  MoveL 3289 to (42.94, 64.74, -221.41) mm, rotated rx 105.8 ry 33.04 rz -145.95 deg; joints [-8.632, -27.169, 98.04, 142.565, 83.685, 20.863, -295]
  MoveL 3290 to (44.16, 62.72, -223.16) mm, rotated rx 105.8 ry 33.04 rz -145.95 deg; joints [-8.699, -27.017, 97.932, 142.503, 83.733, 20.854, -295]
  MoveL 3291 to (44.54, 61.54, -223.78) mm, rotated rx 105.8 ry 33.04 rz -145.95 deg; joints [-8.723, -26.947, 97.904, 142.483, 83.771, 20.834, -295]
  MoveL 3292 to (44.76, 60.25, -224.22) mm, rotated rx 105.8 ry 33.04 rz -145.95 deg; joints [-8.741, -26.881, 97.895, 142.469, 83.82, 20.804, -295]
  MoveL 3293 to (44.72, 57.32, -224.57) mm, rotated rx 105.8 ry 33.04 rz -145.95 deg; joints [-8.758, -26.761, 97.928, 142.462, 83.945, 20.714, -295]
  MoveL 3294 to (44.43, 54.71, -224.56) mm, rotated rx 105.8 ry 33.04 rz -145.95 deg; joints [-8.763, -26.667, 97.984, 142.467, 84.065, 20.624, -295]
  MoveL 3295 to (44.36, 54.19, -224.55) mm, rotated rx 105.8 ry 33.04 rz -145.95 deg; joints [-8.763, -26.649, 97.996, 142.469, 84.089, 20.605, -295]
  MoveL 3296 to (44.28, 53.65, -224.52) mm, rotated rx 105.8 ry 33.04 rz -145.95 deg; joints [-8.763, -26.631, 98.01, 142.471, 84.114, 20.586, -295]
  MoveL 3297 to (44.22, 53.16, -224.51) mm, rotated rx 105.8 ry 33.04 rz -145.95 deg; joints [-8.764, -26.613, 98.021, 142.472, 84.137, 20.568, -295]
  MoveL 3298 to (44.18, 52.72, -224.53) mm, rotated rx 105.8 ry 33.04 rz -145.95 deg; joints [-8.765, -26.597, 98.03, 142.472, 84.157, 20.553, -295]
  MoveL 3299 to (44.14, 52.23, -224.56) mm, rotated rx 105.8 ry 33.04 rz -145.95 deg; joints [-8.767, -26.578, 98.038, 142.472, 84.179, 20.537, -295]
  MoveL 3300 to (44.12, 51.65, -224.63) mm, rotated rx 105.8 ry 33.04 rz -145.95 deg; joints [-8.77, -26.555, 98.046, 142.471, 84.204, 20.519, -295]
  MoveL 3301 to (44.11, 51.07, -224.71) mm, rotated rx 105.8 ry 33.04 rz -145.95 deg; joints [-8.774, -26.531, 98.052, 142.469, 84.229, 20.502, -295]
  MoveL 3302 to (44.08, 50.5, -224.75) mm, rotated rx 105.8 ry 33.04 rz -145.95 deg; joints [-8.777, -26.509, 98.061, 142.468, 84.254, 20.484, -295]
  MoveL 3303 to (44.03, 49.97, -224.78) mm, rotated rx 105.8 ry 33.04 rz -145.95 deg; joints [-8.779, -26.489, 98.07, 142.468, 84.277, 20.466, -295]
  MoveL 3304 to (43.98, 49.46, -224.79) mm, rotated rx 105.8 ry 33.04 rz -145.95 deg; joints [-8.78, -26.47, 98.081, 142.469, 84.301, 20.448, -295]
  MoveL 3305 to (43.92, 48.94, -224.79) mm, rotated rx 105.8 ry 33.04 rz -145.95 deg; joints [-8.781, -26.451, 98.091, 142.47, 84.325, 20.43, -295]
  MoveL 3306 to (43.88, 48.37, -224.82) mm, rotated rx 105.8 ry 33.04 rz -145.95 deg; joints [-8.783, -26.429, 98.101, 142.469, 84.35, 20.412, -295]
  MoveL 3307 to (43.87, 47.82, -224.87) mm, rotated rx 105.8 ry 33.04 rz -145.95 deg; joints [-8.786, -26.407, 98.108, 142.468, 84.374, 20.395, -295]
  MoveL 3308 to (43.87, 47.26, -224.94) mm, rotated rx 105.8 ry 33.04 rz -145.95 deg; joints [-8.789, -26.383, 98.112, 142.467, 84.397, 20.378, -295]
  MoveL 3309 to (43.92, 46.76, -225) mm, rotated rx 105.8 ry 33.04 rz -145.95 deg; joints [-8.792, -26.359, 98.112, 142.465, 84.416, 20.364, -295]
  MoveL 3310 to (44.02, 46.31, -225.03) mm, rotated rx 105.8 ry 33.04 rz -145.95 deg; joints [-8.794, -26.335, 98.107, 142.465, 84.432, 20.353, -295]
  MoveL 3311 to (44.16, 45.93, -225.04) mm, rotated rx 105.8 ry 33.04 rz -145.95 deg; joints [-8.794, -26.311, 98.097, 142.465, 84.442, 20.345, -295]
  MoveL 3312 to (44.32, 45.58, -225.04) mm, rotated rx 105.8 ry 33.04 rz -145.95 deg; joints [-8.794, -26.288, 98.084, 142.466, 84.451, 20.338, -295]
  MoveL 3313 to (43.93, 46.81, -225.92) mm, rotated rx 105.8 ry 33.04 rz -145.95 deg; joints [-8.827, -26.359, 98.105, 142.431, 84.417, 20.377, -295]
  MoveL 3314 to (44.77, 45.44, -226.2) mm, rotated rx 105.8 ry 33.04 rz -145.95 deg; joints [-8.837, -26.257, 98.035, 142.423, 84.444, 20.36, -295]
  MoveL 3315 to (45.67, 43.88, -226.39) mm, rotated rx 105.8 ry 33.04 rz -145.95 deg; joints [-8.845, -26.143, 97.961, 142.418, 84.478, 20.337, -295]
  MoveL 3316 to (46.65, 42.08, -226.52) mm, rotated rx 105.8 ry 33.04 rz -145.95 deg; joints [-8.85, -26.015, 97.882, 142.416, 84.517, 20.309, -295]
  MoveL 3317 to (47.7, 40.09, -226.61) mm, rotated rx 105.8 ry 33.04 rz -145.95 deg; joints [-8.854, -25.875, 97.797, 142.415, 84.562, 20.276, -295]
  MoveL 3318 to (48.71, 38.21, -226.76) mm, rotated rx 105.8 ry 33.04 rz -145.95 deg; joints [-8.86, -25.742, 97.715, 142.412, 84.603, 20.246, -295]
  MoveL 3319 to (49.74, 36.33, -226.97) mm, rotated rx 105.8 ry 33.04 rz -145.95 deg; joints [-8.868, -25.609, 97.631, 142.407, 84.644, 20.218, -295]
  MoveL 3320 to (50.69, 34.54, -227.1) mm, rotated rx 105.8 ry 33.04 rz -145.95 deg; joints [-8.873, -25.482, 97.553, 142.405, 84.683, 20.19, -295]
  MoveL 3321 to (51.59, 32.92, -227.36) mm, rotated rx 105.8 ry 33.04 rz -145.95 deg; joints [-8.883, -25.366, 97.478, 142.397, 84.718, 20.167, -295]
  MoveL 3322 to (52.56, 31.1, -227.58) mm, rotated rx 105.8 ry 33.04 rz -145.95 deg; joints [-8.891, -25.237, 97.397, 142.392, 84.757, 20.14, -295]
  MoveL 3323 to (53.53, 29.26, -227.72) mm, rotated rx 105.8 ry 33.04 rz -145.95 deg; joints [-8.897, -25.108, 97.316, 142.389, 84.797, 20.111, -295]
  MoveL 3324 to (54.52, 27.37, -227.82) mm, rotated rx 105.8 ry 33.04 rz -145.95 deg; joints [-8.901, -24.975, 97.234, 142.388, 84.838, 20.081, -295]
  MoveL 3325 to (55.51, 25.49, -228.05) mm, rotated rx 105.8 ry 33.04 rz -145.95 deg; joints [-8.91, -24.843, 97.151, 142.382, 84.879, 20.053, -295]
  MoveL 3326 to (56.49, 23.58, -228.31) mm, rotated rx 105.8 ry 33.04 rz -145.95 deg; joints [-8.921, -24.709, 97.069, 142.375, 84.921, 20.024, -295]
  MoveL 3327 to (57.47, 21.69, -228.4) mm, rotated rx 105.8 ry 33.04 rz -145.95 deg; joints [-8.924, -24.578, 96.987, 142.374, 84.961, 19.994, -295]
  MoveL 3328 to (58.47, 19.76, -228.44) mm, rotated rx 105.8 ry 33.04 rz -145.95 deg; joints [-8.926, -24.442, 96.903, 142.375, 85.002, 19.963, -295]
  MoveL 3329 to (59.43, 17.88, -228.55) mm, rotated rx 105.8 ry 33.04 rz -145.95 deg; joints [-8.931, -24.311, 96.822, 142.373, 85.042, 19.934, -295]
  MoveL 3330 to (60.39, 15.99, -228.75) mm, rotated rx 105.8 ry 33.04 rz -145.95 deg; joints [-8.939, -24.18, 96.74, 142.368, 85.083, 19.905, -295]
  MoveL 3331 to (61.32, 14.13, -229.08) mm, rotated rx 105.8 ry 33.04 rz -145.95 deg; joints [-8.952, -24.051, 96.66, 142.357, 85.124, 19.879, -295]
  MoveL 3332 to (62.27, 12.2, -229.34) mm, rotated rx 105.8 ry 33.04 rz -145.95 deg; joints [-8.962, -23.918, 96.578, 142.35, 85.167, 19.85, -295]
  MoveL 3333 to (63.21, 10.28, -229.54) mm, rotated rx 105.8 ry 33.04 rz -145.95 deg; joints [-8.97, -23.786, 96.498, 142.345, 85.209, 19.82, -295]
  MoveL 3334 to (64.15, 8.32, -229.78) mm, rotated rx 105.8 ry 33.04 rz -145.95 deg; joints [-8.98, -23.652, 96.416, 142.338, 85.252, 19.79, -295]
  MoveL 3335 to (65.11, 6.4, -229.92) mm, rotated rx 105.8 ry 33.04 rz -145.95 deg; joints [-8.986, -23.519, 96.333, 142.335, 85.293, 19.761, -295]
  MoveL 3336 to (66.08, 4.51, -229.94) mm, rotated rx 105.8 ry 33.04 rz -145.95 deg; joints [-8.987, -23.387, 96.249, 142.336, 85.331, 19.732, -295]
  MoveL 3337 to (65.99, 3.89, -230.61) mm, rotated rx 105.8 ry 33.04 rz -145.95 deg; joints [-9.013, -23.363, 96.257, 142.312, 85.361, 19.718, -295]
  MoveL 3338 to (65.77, 4.13, -230.94) mm, rotated rx 105.8 ry 33.04 rz -145.95 deg; joints [-9.026, -23.385, 96.275, 142.3, 85.361, 19.723, -295]
  MoveL 3339 to (65.73, 4.16, -231.15) mm, rotated rx 105.8 ry 33.04 rz -145.95 deg; joints [-9.034, -23.387, 96.277, 142.292, 85.361, 19.726, -295]
  MoveL 3340 to (65.88, 3.99, -231.25) mm, rotated rx 105.8 ry 33.04 rz -145.95 deg; joints [-9.037, -23.373, 96.264, 142.288, 85.363, 19.726, -295]
  MoveL 3341 to (66.2, 3.72, -231.27) mm, rotated rx 105.8 ry 33.04 rz -145.95 deg; joints [-9.038, -23.344, 96.233, 142.288, 85.362, 19.727, -295]
  MoveC 3342 to (67.05, 3.17, -231.27) mm, rotated rx 105.8 ry 33.04 rz -145.95 deg; joints [-9.036, -23.276, 96.152, 142.289, 85.351, 19.735, -295] to (67.94, 2.68, -231.27) mm, rotated rx 105.8 ry 33.04 rz -145.95 deg; joints [-9.035, -23.209, 96.066, 142.289, 85.336, 19.746, -295]
  MoveL 3343 to (67.94, 2.68, -231.27) mm, rotated rx 105.8 ry 33.04 rz -145.95 deg; joints [-9.035, -23.209, 96.066, 142.289, 85.336, 19.746, -295]
  MoveL 3344 to (68.42, 2.41, -231.3) mm, rotated rx 105.8 ry 33.04 rz -145.95 deg; joints [-9.035, -23.172, 96.021, 142.289, 85.329, 19.751, -295]
  MoveL 3345 to (68.87, 2.12, -231.35) mm, rotated rx 105.8 ry 33.04 rz -145.95 deg; joints [-9.036, -23.136, 95.977, 142.287, 85.323, 19.756, -295]
  MoveL 3346 to (69.36, 1.81, -231.41) mm, rotated rx 105.8 ry 33.04 rz -145.95 deg; joints [-9.038, -23.097, 95.93, 142.285, 85.317, 19.762, -295]
  MoveL 3347 to (69.87, 1.5, -231.46) mm, rotated rx 105.8 ry 33.04 rz -145.95 deg; joints [-9.039, -23.057, 95.881, 142.284, 85.31, 19.767, -295]
  MoveL 3348 to (70.92, 0.9, -231.48) mm, rotated rx 105.8 ry 33.04 rz -145.95 deg; joints [-9.038, -22.976, 95.78, 142.284, 85.293, 19.78, -295]
  MoveL 3349 to (71.4, 0.61, -231.51) mm, rotated rx 105.8 ry 33.04 rz -145.95 deg; joints [-9.038, -22.939, 95.734, 142.283, 85.287, 19.785, -295]
  MoveL 3350 to (71.79, 0.34, -231.58) mm, rotated rx 105.8 ry 33.04 rz -145.95 deg; joints [-9.04, -22.907, 95.696, 142.28, 85.282, 19.789, -295]
  MoveL 3351 to (72.14, 0.08, -231.67) mm, rotated rx 105.8 ry 33.04 rz -145.95 deg; joints [-9.043, -22.878, 95.662, 142.277, 85.279, 19.793, -295]
  MoveL 3352 to (72.5, -0.15, -231.74) mm, rotated rx 105.8 ry 33.04 rz -145.95 deg; joints [-9.045, -22.849, 95.627, 142.275, 85.275, 19.797, -295]
  MoveL 3353 to (72.88, -0.39, -231.77) mm, rotated rx 105.8 ry 33.04 rz -145.95 deg; joints [-9.046, -22.819, 95.59, 142.274, 85.27, 19.801, -295]
  MoveL 3354 to (75.18, -1.65, -231.77) mm, rotated rx 105.8 ry 33.04 rz -145.95 deg; joints [-9.042, -22.645, 95.368, 142.276, 85.231, 19.83, -295]
  MoveL 3355 to (77.59, -3.27, -232.12) mm, rotated rx 105.8 ry 33.04 rz -145.95 deg; joints [-9.051, -22.449, 95.134, 142.265, 85.203, 19.855, -295]
  MoveL 3356 to (78.51, -4.17, -232.55) mm, rotated rx 105.8 ry 33.04 rz -145.95 deg; joints [-9.066, -22.361, 95.044, 142.25, 85.203, 19.861, -295]
  MoveL 3357 to (79.24, -5.11, -233.15) mm, rotated rx 105.8 ry 33.04 rz -145.95 deg; joints [-9.088, -22.281, 94.972, 142.229, 85.213, 19.861, -295]
  MoveL 3358 to (79.79, -6.11, -233.93) mm, rotated rx 105.8 ry 33.04 rz -145.95 deg; joints [-9.118, -22.208, 94.917, 142.201, 85.233, 19.857, -295]
  MoveL 3359 to (80.14, -7.16, -234.88) mm, rotated rx 105.8 ry 33.04 rz -145.95 deg; joints [-9.154, -22.143, 94.88, 142.167, 85.262, 19.848, -295]
  MoveL 3360 to (80.29, -9.41, -237.29) mm, rotated rx 105.8 ry 33.04 rz -145.95 deg; joints [-9.248, -22.033, 94.859, 142.08, 85.35, 19.815, -295]
  MoveL 3361 to (79.77, -11.24, -239.7) mm, rotated rx 105.8 ry 33.04 rz -145.95 deg; joints [-9.343, -21.975, 94.903, 141.992, 85.447, 19.774, -295]
  MoveL 3362 to (79.29, -11.76, -240.65) mm, rotated rx 105.8 ry 33.04 rz -145.95 deg; joints [-9.381, -21.976, 94.947, 141.958, 85.488, 19.756, -295]
  MoveL 3363 to (78.67, -12.02, -241.43) mm, rotated rx 105.8 ry 33.04 rz -145.95 deg; joints [-9.412, -21.996, 95.006, 141.929, 85.524, 19.74, -295]
  MoveL 3364 to (78.3, -12.05, -241.75) mm, rotated rx 105.8 ry 33.04 rz -145.95 deg; joints [-9.425, -22.013, 95.04, 141.917, 85.54, 19.732, -295]
  MoveL 3365 to (77.89, -12.02, -242.03) mm, rotated rx 105.8 ry 33.04 rz -145.95 deg; joints [-9.437, -22.035, 95.079, 141.906, 85.555, 19.724, -295]
  MoveL 3366 to (76.97, -11.75, -242.46) mm, rotated rx 105.8 ry 33.04 rz -145.95 deg; joints [-9.455, -22.093, 95.166, 141.89, 85.582, 19.711, -295]
  MoveL 3367 to (75.9, -11.22, -242.72) mm, rotated rx 105.8 ry 33.04 rz -145.95 deg; joints [-9.467, -22.171, 95.269, 141.879, 85.603, 19.698, -295]
  MoveL 3368 to (74.68, -10.42, -242.81) mm, rotated rx 105.8 ry 33.04 rz -145.95 deg; joints [-9.473, -22.268, 95.386, 141.875, 85.62, 19.687, -295]
  MoveL 3369 to (74.26, -10.12, -242.81) mm, rotated rx 105.8 ry 33.04 rz -145.95 deg; joints [-9.473, -22.304, 95.427, 141.875, 85.624, 19.684, -295]
  MoveL 3370 to (73.91, -9.84, -242.77) mm, rotated rx 105.8 ry 33.04 rz -145.95 deg; joints [-9.473, -22.334, 95.461, 141.875, 85.627, 19.682, -295]
  MoveL 3371 to (73.59, -9.57, -242.72) mm, rotated rx 105.8 ry 33.04 rz -145.95 deg; joints [-9.471, -22.363, 95.491, 141.877, 85.628, 19.68, -295]
  MoveL 3372 to (73.28, -9.29, -242.65) mm, rotated rx 105.8 ry 33.04 rz -145.95 deg; joints [-9.469, -22.39, 95.521, 141.879, 85.629, 19.678, -295]
  MoveL 3373 to (72.94, -9.01, -242.6) mm, rotated rx 105.8 ry 33.04 rz -145.95 deg; joints [-9.468, -22.42, 95.554, 141.881, 85.631, 19.676, -295]
  MoveL 3374 to (72.54, -8.71, -242.58) mm, rotated rx 105.8 ry 33.04 rz -145.95 deg; joints [-9.468, -22.455, 95.593, 141.881, 85.635, 19.673, -295]
  MoveL 3375 to (67.88, -5.36, -242.57) mm, rotated rx 105.8 ry 33.04 rz -145.95 deg; joints [-9.475, -22.84, 96.037, 141.877, 85.683, 19.638, -295]
  MoveL 3376 to (67.27, -4.91, -242.56) mm, rotated rx 105.8 ry 33.04 rz -145.95 deg; joints [-9.476, -22.892, 96.096, 141.876, 85.688, 19.634, -295]
  MoveL 3377 to (66.76, -4.49, -242.55) mm, rotated rx 105.8 ry 33.04 rz -145.95 deg; joints [-9.476, -22.936, 96.144, 141.876, 85.691, 19.632, -295]
  MoveL 3378 to (66.38, -4.06, -242.54) mm, rotated rx 105.8 ry 33.04 rz -145.95 deg; joints [-9.476, -22.975, 96.18, 141.876, 85.689, 19.634, -295]
  MoveL 3379 to (66.07, -3.62, -242.5) mm, rotated rx 105.8 ry 33.04 rz -145.95 deg; joints [-9.475, -23.01, 96.208, 141.877, 85.683, 19.638, -295]
  MoveL 3380 to (65.94, -3.31, -242.34) mm, rotated rx 105.8 ry 33.04 rz -145.95 deg; joints [-9.468, -23.031, 96.221, 141.883, 85.676, 19.641, -295]
  MoveL 3381 to (65.96, -3.3, -242.03) mm, rotated rx 105.8 ry 33.04 rz -145.95 deg; joints [-9.457, -23.031, 96.221, 141.894, 85.674, 19.638, -295]
  MoveL 3382 to (66.15, -3.61, -241.54) mm, rotated rx 105.8 ry 33.04 rz -145.95 deg; joints [-9.438, -23.008, 96.207, 141.913, 85.678, 19.629, -295]
  MoveL 3383 to (66.54, -3.12, -240.57) mm, rotated rx 105.8 ry 33.04 rz -145.95 deg; joints [-9.4, -23.011, 96.173, 141.949, 85.641, 19.643, -295]
  MoveL 3384 to (65.93, -1.35, -240.27) mm, rotated rx 105.8 ry 33.04 rz -145.95 deg; joints [-9.387, -23.12, 96.225, 141.958, 85.595, 19.675, -295]
  MoveL 3385 to (65.28, 0.49, -240.07) mm, rotated rx 105.8 ry 33.04 rz -145.95 deg; joints [-9.378, -23.235, 96.281, 141.964, 85.546, 19.71, -295]
  MoveL 3386 to (64.55, 2.49, -239.94) mm, rotated rx 105.8 ry 33.04 rz -145.95 deg; joints [-9.372, -23.36, 96.341, 141.967, 85.495, 19.748, -295]
  MoveL 3387 to (63.05, 6.49, -239.94) mm, rotated rx 105.8 ry 33.04 rz -145.95 deg; joints [-9.37, -23.611, 96.463, 141.962, 85.393, 19.827, -295]
  MoveL 3388 to (62.36, 8.35, -239.85) mm, rotated rx 105.8 ry 33.04 rz -145.95 deg; joints [-9.365, -23.727, 96.52, 141.964, 85.345, 19.863, -295]
  MoveL 3389 to (61.61, 10.35, -239.85) mm, rotated rx 105.8 ry 33.04 rz -145.95 deg; joints [-9.364, -23.852, 96.58, 141.962, 85.293, 19.903, -295]
  MoveL 3390 to (60.95, 12.4, -239.85) mm, rotated rx 105.8 ry 33.04 rz -145.95 deg; joints [-9.363, -23.975, 96.631, 141.959, 85.236, 19.947, -295]
  MoveL 3391 to (60.21, 14.84, -239.67) mm, rotated rx 105.8 ry 33.04 rz -145.95 deg; joints [-9.354, -24.119, 96.688, 141.963, 85.166, 19.999, -295]
  MoveL 3392 to (59.31, 16.87, -239.44) mm, rotated rx 105.8 ry 33.04 rz -145.95 deg; joints [-9.345, -24.254, 96.763, 141.969, 85.118, 20.033, -295]
  MoveL 3393 to (58.46, 18.87, -239.32) mm, rotated rx 105.8 ry 33.04 rz -145.95 deg; joints [-9.339, -24.384, 96.833, 141.972, 85.069, 20.07, -295]
  MoveL 3394 to (57.71, 20.87, -239.21) mm, rotated rx 105.8 ry 33.04 rz -145.95 deg; joints [-9.334, -24.509, 96.892, 141.973, 85.016, 20.109, -295]
  MoveL 3395 to (56.95, 22.87, -239) mm, rotated rx 105.8 ry 33.04 rz -145.95 deg; joints [-9.325, -24.634, 96.952, 141.979, 84.963, 20.147, -295]
  MoveL 3396 to (56.2, 24.86, -238.89) mm, rotated rx 105.8 ry 33.04 rz -145.95 deg; joints [-9.32, -24.759, 97.011, 141.98, 84.91, 20.187, -295]
  MoveL 3397 to (55.44, 26.86, -238.78) mm, rotated rx 105.8 ry 33.04 rz -145.95 deg; joints [-9.314, -24.884, 97.07, 141.981, 84.857, 20.227, -295]
  MoveL 3398 to (54.68, 28.85, -238.57) mm, rotated rx 105.8 ry 33.04 rz -145.95 deg; joints [-9.305, -25.01, 97.13, 141.987, 84.804, 20.265, -295]
  MoveL 3399 to (53.92, 30.84, -238.46) mm, rotated rx 105.8 ry 33.04 rz -145.95 deg; joints [-9.3, -25.135, 97.188, 141.988, 84.75, 20.305, -295]
  MoveL 3400 to (53.16, 32.83, -238.36) mm, rotated rx 105.8 ry 33.04 rz -145.95 deg; joints [-9.295, -25.259, 97.246, 141.989, 84.697, 20.345, -295]
  MoveL 3401 to (52.38, 34.82, -238.15) mm, rotated rx 105.8 ry 33.04 rz -145.95 deg; joints [-9.286, -25.385, 97.307, 141.994, 84.644, 20.383, -295]
  MoveL 3402 to (51.61, 36.81, -238.05) mm, rotated rx 105.8 ry 33.04 rz -145.95 deg; joints [-9.281, -25.51, 97.364, 141.995, 84.59, 20.423, -295]
  MoveL 3403 to (50.88, 38.51, -237.79) mm, rotated rx 105.8 ry 33.04 rz -145.95 deg; joints [-9.271, -25.621, 97.422, 142.002, 84.546, 20.453, -295]
  MoveL 3404 to (50.16, 40.02, -237.43) mm, rotated rx 105.8 ry 33.04 rz -145.95 deg; joints [-9.257, -25.723, 97.481, 142.013, 84.509, 20.477, -295]
  MoveL 3405 to (49.44, 41.36, -236.92) mm, rotated rx 105.8 ry 33.04 rz -145.95 deg; joints [-9.238, -25.818, 97.542, 142.03, 84.479, 20.493, -295]
  MoveL 3406 to (49.6, 40.24, -236.08) mm, rotated rx 105.8 ry 33.04 rz -145.95 deg; joints [-9.207, -25.764, 97.544, 142.063, 84.517, 20.451, -295]
  MoveL 3407 to (49.48, 40.55, -236.05) mm, rotated rx 105.8 ry 33.04 rz -145.95 deg; joints [-9.206, -25.783, 97.552, 142.063, 84.508, 20.457, -295]
  MoveL 3408 to (49.4, 40.86, -236.01) mm, rotated rx 105.8 ry 33.04 rz -145.95 deg; joints [-9.204, -25.801, 97.558, 142.065, 84.498, 20.464, -295]
  MoveL 3409 to (49.39, 41.23, -235.95) mm, rotated rx 105.8 ry 33.04 rz -145.95 deg; joints [-9.201, -25.817, 97.556, 142.066, 84.483, 20.475, -295]
  MoveL 3410 to (49.43, 41.65, -235.92) mm, rotated rx 105.8 ry 33.04 rz -145.95 deg; joints [-9.199, -25.833, 97.549, 142.067, 84.464, 20.489, -295]
  MoveL 3411 to (49.51, 42.12, -235.89) mm, rotated rx 105.8 ry 33.04 rz -145.95 deg; joints [-9.197, -25.849, 97.536, 142.067, 84.442, 20.506, -295]
  MoveL 3412 to (50.6, 46.71, -235.89) mm, rotated rx 105.8 ry 33.04 rz -145.95 deg; joints [-9.187, -25.985, 97.385, 142.059, 84.214, 20.68, -295]
  MoveL 3413 to (50.67, 47.11, -235.87) mm, rotated rx 105.8 ry 33.04 rz -145.95 deg; joints [-9.185, -25.997, 97.374, 142.059, 84.195, 20.694, -295]
  MoveL 3414 to (50.79, 47.61, -235.87) mm, rotated rx 105.8 ry 33.04 rz -145.95 deg; joints [-9.184, -26.012, 97.358, 142.059, 84.169, 20.714, -295]
  MoveL 3415 to (51, 48.62, -235.83) mm, rotated rx 105.8 ry 33.04 rz -145.95 deg; joints [-9.181, -26.043, 97.327, 142.058, 84.12, 20.751, -295]
  MoveL 3416 to (51.61, 51.17, -235.83) mm, rotated rx 105.8 ry 33.04 rz -145.95 deg; joints [-9.175, -26.118, 97.242, 142.053, 83.993, 20.848, -295]
  MoveL 3417 to (51.79, 52.19, -235.81) mm, rotated rx 105.8 ry 33.04 rz -145.95 deg; joints [-9.172, -26.151, 97.214, 142.052, 83.945, 20.885, -295]
  MoveL 3418 to (52.1, 53.6, -235.87) mm, rotated rx 105.8 ry 33.04 rz -145.95 deg; joints [-9.172, -26.192, 97.168, 142.047, 83.875, 20.939, -295]
  MoveL 3419 to (52.5, 54.7, -236.13) mm, rotated rx 105.8 ry 33.04 rz -145.95 deg; joints [-9.179, -26.217, 97.116, 142.035, 83.816, 20.988, -295]
  MoveL 3420 to (52.97, 55.5, -236.57) mm, rotated rx 105.8 ry 33.04 rz -145.95 deg; joints [-9.193, -26.224, 97.058, 142.017, 83.768, 21.032, -295]
  MoveL 3421 to (53.23, 55.79, -236.86) mm, rotated rx 105.8 ry 33.04 rz -145.95 deg; joints [-9.202, -26.221, 97.026, 142.006, 83.748, 21.052, -295]
  MoveL 3422 to (53.52, 55.99, -237.19) mm, rotated rx 105.8 ry 33.04 rz -145.95 deg; joints [-9.214, -26.213, 96.994, 141.993, 83.73, 21.071, -295]
  MoveL 3423 to (54.15, 56.18, -238.01) mm, rotated rx 105.8 ry 33.04 rz -145.95 deg; joints [-9.242, -26.186, 96.924, 141.962, 83.702, 21.105, -295]
  MoveL 3424 to (54.86, 56.07, -239) mm, rotated rx 105.8 ry 33.04 rz -145.95 deg; joints [-9.278, -26.141, 96.848, 141.925, 83.685, 21.133, -295]
  MoveL 3425 to (56.51, 54.91, -241.56) mm, rotated rx 105.8 ry 33.04 rz -145.95 deg; joints [-9.371, -26, 96.678, 141.833, 83.682, 21.176, -295]
  MoveL 3426 to (57.96, 53, -244.13) mm, rotated rx 105.8 ry 33.04 rz -145.95 deg; joints [-9.467, -25.838, 96.536, 141.741, 83.717, 21.188, -295]
  MoveL 3427 to (58.68, 50.78, -245.96) mm, rotated rx 105.8 ry 33.04 rz -145.95 deg; joints [-9.537, -25.704, 96.473, 141.678, 83.787, 21.162, -295]
  MoveL 3428 to (58.77, 49.56, -246.6) mm, rotated rx 105.8 ry 33.04 rz -145.95 deg; joints [-9.563, -25.647, 96.472, 141.657, 83.836, 21.134, -295]
  MoveL 3429 to (58.68, 48.26, -247.06) mm, rotated rx 105.8 ry 33.04 rz -145.95 deg; joints [-9.582, -25.597, 96.49, 141.642, 83.894, 21.096, -295]
  MoveL 3430 to (57.95, 45.43, -247.42) mm, rotated rx 105.8 ry 33.04 rz -145.95 deg; joints [-9.603, -25.517, 96.587, 141.634, 84.037, 20.991, -295]
  MoveL 3431 to (56.87, 42.48, -247.42) mm, rotated rx 105.8 ry 33.04 rz -145.95 deg; joints [-9.611, -25.451, 96.722, 141.639, 84.196, 20.868, -295]
  MoveL 3432 to (56.54, 41.51, -247.44) mm, rotated rx 105.8 ry 33.04 rz -145.95 deg; joints [-9.614, -25.428, 96.763, 141.64, 84.247, 20.828, -295]
  MoveL 3433 to (56.18, 40.53, -247.44) mm, rotated rx 105.8 ry 33.04 rz -145.95 deg; joints [-9.616, -25.406, 96.808, 141.641, 84.3, 20.787, -295]
  MoveL 3434 to (56.01, 40.06, -247.44) mm, rotated rx 105.8 ry 33.04 rz -145.95 deg; joints [-9.618, -25.395, 96.829, 141.642, 84.325, 20.768, -295]
  MoveL 3435 to (55.8, 39.43, -247.47) mm, rotated rx 105.8 ry 33.04 rz -145.95 deg; joints [-9.621, -25.38, 96.856, 141.642, 84.358, 20.742, -295]
  MoveL 3436 to (55.62, 38.86, -247.53) mm, rotated rx 105.8 ry 33.04 rz -145.95 deg; joints [-9.624, -25.365, 96.878, 141.641, 84.388, 20.72, -295]
  MoveL 3437 to (55.49, 38.38, -247.6) mm, rotated rx 105.8 ry 33.04 rz -145.95 deg; joints [-9.628, -25.351, 96.895, 141.639, 84.413, 20.702, -295]
  MoveL 3438 to (55.36, 37.93, -247.65) mm, rotated rx 105.8 ry 33.04 rz -145.95 deg; joints [-9.631, -25.339, 96.911, 141.637, 84.436, 20.685, -295]
  MoveL 3439 to (55.22, 37.49, -247.69) mm, rotated rx 105.8 ry 33.04 rz -145.95 deg; joints [-9.634, -25.328, 96.929, 141.637, 84.459, 20.668, -295]
  MoveL 3440 to (54.68, 36.01, -247.69) mm, rotated rx 105.8 ry 33.04 rz -145.95 deg; joints [-9.638, -25.294, 96.995, 141.639, 84.539, 20.606, -295]
  MoveL 3441 to (54.53, 35.53, -247.7) mm, rotated rx 105.8 ry 33.04 rz -145.95 deg; joints [-9.64, -25.282, 97.015, 141.639, 84.564, 20.587, -295]
  MoveL 3442 to (54.42, 35.11, -247.73) mm, rotated rx 105.8 ry 33.04 rz -145.95 deg; joints [-9.642, -25.27, 97.029, 141.638, 84.585, 20.571, -295]
  MoveL 3443 to (54.35, 34.73, -247.77) mm, rotated rx 105.8 ry 33.04 rz -145.95 deg; joints [-9.644, -25.257, 97.039, 141.637, 84.603, 20.557, -295]
  MoveL 3444 to (54.36, 34.42, -247.84) mm, rotated rx 105.8 ry 33.04 rz -145.95 deg; joints [-9.647, -25.243, 97.04, 141.635, 84.615, 20.549, -295]
  MoveL 3445 to (54.41, 34.15, -247.91) mm, rotated rx 105.8 ry 33.04 rz -145.95 deg; joints [-9.65, -25.229, 97.037, 141.633, 84.624, 20.543, -295]
  MoveL 3446 to (54.73, 35.71, -248.71) mm, rotated rx 105.8 ry 33.04 rz -145.95 deg; joints [-9.677, -25.276, 96.985, 141.601, 84.552, 20.611, -295]
  MoveL 3447 to (55.11, 33.98, -249.12) mm, rotated rx 105.8 ry 33.04 rz -145.95 deg; joints [-9.694, -25.183, 96.96, 141.589, 84.609, 20.573, -295]
  MoveL 3448 to (55.54, 32.16, -249.38) mm, rotated rx 105.8 ry 33.04 rz -145.95 deg; joints [-9.706, -25.082, 96.931, 141.582, 84.668, 20.531, -295]
  MoveL 3449 to (56.03, 30.22, -249.56) mm, rotated rx 105.8 ry 33.04 rz -145.95 deg; joints [-9.714, -24.974, 96.899, 141.577, 84.729, 20.485, -295]
  MoveL 3450 to (56.57, 28.16, -249.76) mm, rotated rx 105.8 ry 33.04 rz -145.95 deg; joints [-9.724, -24.857, 96.862, 141.573, 84.793, 20.438, -295]
  MoveL 3451 to (57.09, 26.08, -249.85) mm, rotated rx 105.8 ry 33.04 rz -145.95 deg; joints [-9.729, -24.742, 96.827, 141.572, 84.857, 20.389, -295]
  MoveL 3452 to (57.61, 24.02, -249.95) mm, rotated rx 105.8 ry 33.04 rz -145.95 deg; joints [-9.735, -24.626, 96.792, 141.571, 84.921, 20.34, -295]
  MoveL 3453 to (58.14, 21.95, -250.15) mm, rotated rx 105.8 ry 33.04 rz -145.95 deg; joints [-9.744, -24.51, 96.755, 141.566, 84.985, 20.293, -295]
  MoveL 3454 to (58.66, 19.88, -250.25) mm, rotated rx 105.8 ry 33.04 rz -145.95 deg; joints [-9.75, -24.394, 96.719, 141.565, 85.049, 20.244, -295]
  MoveL 3455 to (59.17, 17.81, -250.35) mm, rotated rx 105.8 ry 33.04 rz -145.95 deg; joints [-9.756, -24.278, 96.684, 141.564, 85.113, 20.196, -295]
  MoveL 3456 to (59.69, 15.74, -250.55) mm, rotated rx 105.8 ry 33.04 rz -145.95 deg; joints [-9.765, -24.162, 96.647, 141.559, 85.177, 20.148, -295]
  MoveL 3457 to (60.71, 11.59, -250.75) mm, rotated rx 105.8 ry 33.04 rz -145.95 deg; joints [-9.777, -23.93, 96.575, 141.556, 85.304, 20.051, -295]
  MoveL 3458 to (61.13, 9.85, -250.96) mm, rotated rx 105.8 ry 33.04 rz -145.95 deg; joints [-9.786, -23.832, 96.543, 141.55, 85.358, 20.012, -295]
  MoveL 3459 to (61.63, 7.95, -251.03) mm, rotated rx 105.8 ry 33.04 rz -145.95 deg; joints [-9.791, -23.724, 96.506, 141.549, 85.414, 19.969, -295]
  MoveL 3460 to (62.22, 5.98, -251.04) mm, rotated rx 105.8 ry 33.04 rz -145.95 deg; joints [-9.793, -23.609, 96.462, 141.55, 85.47, 19.925, -295]
  MoveL 3461 to (62.84, 3.38, -251.15) mm, rotated rx 105.8 ry 33.04 rz -145.95 deg; joints [-9.8, -23.464, 96.416, 141.549, 85.549, 19.865, -295]
  MoveL 3462 to (63.33, 0.85, -251.24) mm, rotated rx 105.8 ry 33.04 rz -145.95 deg; joints [-9.806, -23.328, 96.383, 141.547, 85.63, 19.802, -295]
  MoveL 3463 to (63.81, -1.31, -251.34) mm, rotated rx 105.8 ry 33.04 rz -145.95 deg; joints [-9.812, -23.209, 96.348, 141.546, 85.697, 19.751, -295]
  MoveL 3464 to (64.27, -3.3, -251.51) mm, rotated rx 105.8 ry 33.04 rz -145.95 deg; joints [-9.82, -23.098, 96.312, 141.541, 85.758, 19.706, -295]
  MoveL 3465 to (64.69, -5.16, -251.79) mm, rotated rx 105.8 ry 33.04 rz -145.95 deg; joints [-9.833, -22.995, 96.279, 141.532, 85.815, 19.665, -295]
  MoveL 3466 to (65.1, -7.01, -252.08) mm, rotated rx 105.8 ry 33.04 rz -145.95 deg; joints [-9.846, -22.892, 96.247, 141.523, 85.872, 19.624, -295]
  MoveL 3467 to (65.48, -8.85, -252.37) mm, rotated rx 105.8 ry 33.04 rz -145.95 deg; joints [-9.859, -22.791, 96.217, 141.513, 85.931, 19.583, -295]
  MoveL 3468 to (65.91, -10.79, -252.53) mm, rotated rx 105.8 ry 33.04 rz -145.95 deg; joints [-9.867, -22.684, 96.183, 141.508, 85.99, 19.539, -295]
  MoveL 3469 to (65.58, -11.35, -253.15) mm, rotated rx 105.8 ry 33.04 rz -145.95 deg; joints [-9.892, -22.675, 96.214, 141.485, 86.025, 19.52, -295]
  MoveL 3470 to (65.37, -11.11, -253.46) mm, rotated rx 105.8 ry 33.04 rz -145.95 deg; joints [-9.904, -22.695, 96.23, 141.473, 86.024, 19.525, -295]
  MoveL 3471 to (65.33, -11.11, -253.65) mm, rotated rx 105.8 ry 33.04 rz -145.95 deg; joints [-9.912, -22.697, 96.233, 141.466, 86.027, 19.526, -295]
  MoveL 3472 to (65.44, -11.34, -253.75) mm, rotated rx 105.8 ry 33.04 rz -145.95 deg; joints [-9.915, -22.681, 96.223, 141.463, 86.031, 19.523, -295]
  MoveL 3473 to (65.7, -11.7, -253.77) mm, rotated rx 105.8 ry 33.04 rz -145.95 deg; joints [-9.916, -22.652, 96.198, 141.463, 86.035, 19.52, -295]
  MoveL 3474 to (66.02, -12.07, -253.77) mm, rotated rx 105.8 ry 33.04 rz -145.95 deg; joints [-9.916, -22.619, 96.168, 141.463, 86.037, 19.519, -295]
  MoveL 3475 to (66.74, -12.73, -253.8) mm, rotated rx 105.8 ry 33.04 rz -145.95 deg; joints [-9.916, -22.553, 96.1, 141.463, 86.036, 19.52, -295]
  MoveL 3476 to (67.9, -13.79, -253.8) mm, rotated rx 105.8 ry 33.04 rz -145.95 deg; joints [-9.914, -22.447, 95.99, 141.464, 86.032, 19.522, -295]
  MoveL 3477 to (68.6, -14.48, -253.82) mm, rotated rx 105.8 ry 33.04 rz -145.95 deg; joints [-9.914, -22.381, 95.924, 141.465, 86.032, 19.522, -295]
  MoveL 3478 to (69.37, -15.18, -253.82) mm, rotated rx 105.8 ry 33.04 rz -145.95 deg; joints [-9.913, -22.31, 95.851, 141.466, 86.03, 19.523, -295]
  MoveL 3479 to (69.75, -15.54, -253.84) mm, rotated rx 105.8 ry 33.04 rz -145.95 deg; joints [-9.913, -22.275, 95.815, 141.466, 86.029, 19.524, -295]
  MoveL 3480 to (70.09, -15.87, -253.86) mm, rotated rx 105.8 ry 33.04 rz -145.95 deg; joints [-9.913, -22.244, 95.783, 141.465, 86.029, 19.524, -295]
  MoveL 3481 to (70.4, -16.18, -253.91) mm, rotated rx 105.8 ry 33.04 rz -145.95 deg; joints [-9.915, -22.214, 95.753, 141.464, 86.029, 19.525, -295]
  MoveL 3482 to (70.67, -16.47, -253.97) mm, rotated rx 105.8 ry 33.04 rz -145.95 deg; joints [-9.917, -22.187, 95.726, 141.462, 86.03, 19.525, -295]
  MoveL 3483 to (70.96, -16.77, -254.03) mm, rotated rx 105.8 ry 33.04 rz -145.95 deg; joints [-9.918, -22.158, 95.698, 141.46, 86.03, 19.525, -295]
  MoveL 3484 to (71.29, -17.1, -254.06) mm, rotated rx 105.8 ry 33.04 rz -145.95 deg; joints [-9.919, -22.127, 95.667, 141.459, 86.03, 19.525, -295]
  MoveL 3485 to (71.64, -17.43, -254.08) mm, rotated rx 105.8 ry 33.04 rz -145.95 deg; joints [-9.92, -22.095, 95.634, 141.459, 86.03, 19.526, -295]
  MoveL 3486 to (71.94, -17.74, -254.13) mm, rotated rx 105.8 ry 33.04 rz -145.95 deg; joints [-9.921, -22.065, 95.605, 141.458, 86.03, 19.526, -295]
  MoveL 3487 to (72.21, -18.04, -254.19) mm, rotated rx 105.8 ry 33.04 rz -145.95 deg; joints [-9.923, -22.038, 95.579, 141.456, 86.032, 19.525, -295]
  MoveL 3488 to (72.48, -18.34, -254.24) mm, rotated rx 105.8 ry 33.04 rz -145.95 deg; joints [-9.924, -22.011, 95.552, 141.454, 86.033, 19.525, -295]
  MoveL 3489 to (72.8, -18.66, -254.27) mm, rotated rx 105.8 ry 33.04 rz -145.95 deg; joints [-9.925, -21.981, 95.522, 141.454, 86.033, 19.525, -295]
  MoveL 3490 to (73.18, -19.01, -254.27) mm, rotated rx 105.8 ry 33.04 rz -145.95 deg; joints [-9.924, -21.945, 95.485, 141.454, 86.031, 19.526, -295]
  MoveL 3491 to (75.16, -21.16, -254.63) mm, rotated rx 105.8 ry 33.04 rz -145.95 deg; joints [-9.935, -21.749, 95.295, 141.444, 86.038, 19.525, -295]
  MoveL 3492 to (75.86, -22.24, -255.07) mm, rotated rx 105.8 ry 33.04 rz -145.95 deg; joints [-9.952, -21.664, 95.225, 141.428, 86.052, 19.52, -295]
  MoveL 3493 to (76.39, -23.31, -255.69) mm, rotated rx 105.8 ry 33.04 rz -145.95 deg; joints [-9.976, -21.588, 95.172, 141.406, 86.074, 19.511, -295]
  MoveL 3494 to (76.88, -25.48, -257.48) mm, rotated rx 105.8 ry 33.04 rz -145.95 deg; joints [-10.045, -21.464, 95.116, 141.341, 86.14, 19.483, -295]
  MoveL 3495 to (76.63, -27.66, -259.97) mm, rotated rx 105.8 ry 33.04 rz -145.95 deg; joints [-10.144, -21.375, 95.128, 141.249, 86.237, 19.441, -295]
  MoveL 3496 to (75.82, -29.26, -262.46) mm, rotated rx 105.8 ry 33.04 rz -145.95 deg; joints [-10.244, -21.339, 95.193, 141.156, 86.332, 19.4, -295]
  MoveL 3497 to (75.28, -29.64, -263.44) mm, rotated rx 105.8 ry 33.04 rz -145.95 deg; joints [-10.283, -21.348, 95.239, 141.119, 86.369, 19.385, -295]
  MoveL 3498 to (74.65, -29.73, -264.24) mm, rotated rx 105.8 ry 33.04 rz -145.95 deg; joints [-10.316, -21.374, 95.296, 141.088, 86.398, 19.373, -295]
  MoveL 3499 to (74.3, -29.67, -264.58) mm, rotated rx 105.8 ry 33.04 rz -145.95 deg; joints [-10.33, -21.394, 95.327, 141.076, 86.409, 19.368, -295]
  MoveL 3500 to (73.93, -29.53, -264.87) mm, rotated rx 105.8 ry 33.04 rz -145.95 deg; joints [-10.342, -21.418, 95.362, 141.064, 86.419, 19.365, -295]
  MoveL 3501 to (73.11, -29.05, -265.31) mm, rotated rx 105.8 ry 33.04 rz -145.95 deg; joints [-10.36, -21.48, 95.437, 141.047, 86.433, 19.36, -295]
  MoveL 3502 to (72.21, -28.28, -265.58) mm, rotated rx 105.8 ry 33.04 rz -145.95 deg; joints [-10.372, -21.56, 95.522, 141.035, 86.439, 19.359, -295]
  MoveL 3503 to (71.21, -27.23, -265.67) mm, rotated rx 105.8 ry 33.04 rz -145.95 deg; joints [-10.377, -21.657, 95.617, 141.031, 86.438, 19.362, -295]
  MoveL 3504 to (69.49, -25.25, -265.67) mm, rotated rx 105.8 ry 33.04 rz -145.95 deg; joints [-10.379, -21.832, 95.78, 141.028, 86.429, 19.37, -295]
  MoveL 3505 to (69.21, -24.91, -265.64) mm, rotated rx 105.8 ry 33.04 rz -145.95 deg; joints [-10.378, -21.862, 95.807, 141.029, 86.427, 19.371, -295]
  MoveL 3506 to (68.97, -24.59, -265.59) mm, rotated rx 105.8 ry 33.04 rz -145.95 deg; joints [-10.376, -21.889, 95.83, 141.03, 86.424, 19.373, -295]
  MoveL 3507 to (68.74, -24.28, -265.52) mm, rotated rx 105.8 ry 33.04 rz -145.95 deg; joints [-10.374, -21.914, 95.852, 141.032, 86.421, 19.375, -295]
  MoveL 3508 to (68.48, -23.94, -265.47) mm, rotated rx 105.8 ry 33.04 rz -145.95 deg; joints [-10.372, -21.943, 95.877, 141.034, 86.418, 19.377, -295]
  MoveL 3509 to (68.16, -23.55, -265.43) mm, rotated rx 105.8 ry 33.04 rz -145.95 deg; joints [-10.371, -21.976, 95.907, 141.035, 86.415, 19.379, -295]
  MoveL 3510 to (67.84, -23.13, -265.37) mm, rotated rx 105.8 ry 33.04 rz -145.95 deg; joints [-10.369, -22.011, 95.938, 141.036, 86.411, 19.381, -295]
  MoveL 3511 to (67.49, -22.72, -265.36) mm, rotated rx 105.8 ry 33.04 rz -145.95 deg; joints [-10.369, -22.047, 95.971, 141.037, 86.409, 19.383, -295]
  MoveL 3512 to (67.07, -22.24, -265.37) mm, rotated rx 105.8 ry 33.04 rz -145.95 deg; joints [-10.37, -22.09, 96.011, 141.035, 86.407, 19.385, -295]
  MoveL 3513 to (66.48, -21.6, -265.44) mm, rotated rx 105.8 ry 33.04 rz -145.95 deg; joints [-10.374, -22.148, 96.066, 141.032, 86.405, 19.387, -295]
  MoveL 3514 to (66.13, -21.2, -265.44) mm, rotated rx 105.8 ry 33.04 rz -145.95 deg; joints [-10.374, -22.183, 96.099, 141.031, 86.403, 19.389, -295]
  MoveL 3515 to (65.81, -20.83, -265.43) mm, rotated rx 105.8 ry 33.04 rz -145.95 deg; joints [-10.374, -22.217, 96.129, 141.031, 86.401, 19.391, -295]
  MoveL 3516 to (65.51, -20.47, -265.41) mm, rotated rx 105.8 ry 33.04 rz -145.95 deg; joints [-10.374, -22.248, 96.158, 141.032, 86.399, 19.393, -295]
  MoveL 3517 to (65.26, -20.14, -265.36) mm, rotated rx 105.8 ry 33.04 rz -145.95 deg; joints [-10.372, -22.276, 96.182, 141.033, 86.396, 19.395, -295]
  MoveL 3518 to (65.03, -19.81, -265.3) mm, rotated rx 105.8 ry 33.04 rz -145.95 deg; joints [-10.37, -22.302, 96.203, 141.035, 86.392, 19.397, -295]
  MoveL 3519 to (64.83, -19.44, -265.25) mm, rotated rx 105.8 ry 33.04 rz -145.95 deg; joints [-10.368, -22.329, 96.222, 141.036, 86.385, 19.402, -295]
  MoveL 3520 to (64.67, -19.06, -265.19) mm, rotated rx 105.8 ry 33.04 rz -145.95 deg; joints [-10.366, -22.354, 96.237, 141.038, 86.376, 19.408, -295]
  MoveL 3521 to (64.64, -18.84, -265.03) mm, rotated rx 105.8 ry 33.04 rz -145.95 deg; joints [-10.359, -22.365, 96.24, 141.044, 86.369, 19.412, -295]
  MoveL 3522 to (64.74, -18.89, -264.72) mm, rotated rx 105.8 ry 33.04 rz -145.95 deg; joints [-10.347, -22.359, 96.233, 141.056, 86.367, 19.409, -295]
  MoveL 3523 to (64.97, -19.26, -264.23) mm, rotated rx 105.8 ry 33.04 rz -145.95 deg; joints [-10.328, -22.332, 96.216, 141.075, 86.371, 19.399, -295]
  MoveL 3524 to (64.83, -18.38, -263.37) mm, rotated rx 105.8 ry 33.04 rz -145.95 deg; joints [-10.295, -22.38, 96.234, 141.106, 86.342, 19.41, -295]
  MoveL 3525 to (64.29, -14.15, -263.37) mm, rotated rx 105.8 ry 33.04 rz -145.95 deg; joints [-10.289, -22.594, 96.267, 141.105, 86.2, 19.523, -295]
  MoveL 3526 to (64.04, -12.17, -263.31) mm, rotated rx 105.8 ry 33.04 rz -145.95 deg; joints [-10.284, -22.694, 96.282, 141.106, 86.132, 19.576, -295]
  MoveL 3527 to (63.81, -10.19, -263.16) mm, rotated rx 105.8 ry 33.04 rz -145.95 deg; joints [-10.275, -22.794, 96.296, 141.111, 86.064, 19.628, -295]
  MoveL 3528 to (63.54, -7.91, -262.96) mm, rotated rx 105.8 ry 33.04 rz -145.95 deg; joints [-10.264, -22.908, 96.312, 141.117, 85.986, 19.687, -295]
  MoveL 3529 to (63.28, -5.75, -262.75) mm, rotated rx 105.8 ry 33.04 rz -145.95 deg; joints [-10.253, -23.016, 96.327, 141.124, 85.912, 19.743, -295]
  MoveL 3530 to (63.02, -3.59, -262.65) mm, rotated rx 105.8 ry 33.04 rz -145.95 deg; joints [-10.246, -23.125, 96.342, 141.126, 85.837, 19.8, -295]
  MoveL 3531 to (62.75, -1.47, -262.65) mm, rotated rx 105.8 ry 33.04 rz -145.95 deg; joints [-10.243, -23.231, 96.356, 141.125, 85.765, 19.858, -295]
  MoveL 3532 to (62.49, 0.5, -262.58) mm, rotated rx 105.8 ry 33.04 rz -145.95 deg; joints [-10.238, -23.33, 96.37, 141.126, 85.698, 19.91, -295]
  MoveL 3533 to (62.25, 2.36, -262.47) mm, rotated rx 105.8 ry 33.04 rz -145.95 deg; joints [-10.231, -23.423, 96.383, 141.129, 85.634, 19.959, -295]
  MoveL 3534 to (61.99, 4.38, -262.4) mm, rotated rx 105.8 ry 33.04 rz -145.95 deg; joints [-10.226, -23.525, 96.396, 141.13, 85.564, 20.014, -295]
  MoveL 3535 to (61.72, 6.5, -262.22) mm, rotated rx 105.8 ry 33.04 rz -145.95 deg; joints [-10.216, -23.631, 96.411, 141.135, 85.491, 20.069, -295]
  MoveL 3536 to (61.18, 10.73, -262.04) mm, rotated rx 105.8 ry 33.04 rz -145.95 deg; joints [-10.203, -23.842, 96.437, 141.138, 85.345, 20.182, -295]
  MoveL 3537 to (60.89, 12.85, -261.86) mm, rotated rx 105.8 ry 33.04 rz -145.95 deg; joints [-10.193, -23.949, 96.451, 141.143, 85.271, 20.238, -295]
  MoveL 3538 to (60.61, 14.97, -261.68) mm, rotated rx 105.8 ry 33.04 rz -145.95 deg; joints [-10.184, -24.055, 96.466, 141.148, 85.198, 20.293, -295]
  MoveL 3539 to (60.34, 17.08, -261.68) mm, rotated rx 105.8 ry 33.04 rz -145.95 deg; joints [-10.181, -24.16, 96.477, 141.145, 85.124, 20.352, -295]
  MoveL 3540 to (60.05, 19.2, -261.5) mm, rotated rx 105.8 ry 33.04 rz -145.95 deg; joints [-10.171, -24.266, 96.491, 141.15, 85.051, 20.408, -295]
  MoveL 3541 to (59.75, 21.31, -261.32) mm, rotated rx 105.8 ry 33.04 rz -145.95 deg; joints [-10.162, -24.372, 96.505, 141.154, 84.977, 20.463, -295]
  MoveL 3542 to (59.48, 23.43, -261.32) mm, rotated rx 105.8 ry 33.04 rz -145.95 deg; joints [-10.159, -24.476, 96.515, 141.152, 84.903, 20.522, -295]
  MoveL 3543 to (59.16, 25.35, -261.13) mm, rotated rx 105.8 ry 33.04 rz -145.95 deg; joints [-10.149, -24.575, 96.532, 141.157, 84.838, 20.571, -295]
  MoveL 3544 to (58.82, 27.03, -260.81) mm, rotated rx 105.8 ry 33.04 rz -145.95 deg; joints [-10.135, -24.665, 96.555, 141.166, 84.783, 20.61, -295]
  MoveL 3545 to (58.43, 28.51, -260.34) mm, rotated rx 105.8 ry 33.04 rz -145.95 deg; joints [-10.116, -24.75, 96.585, 141.182, 84.737, 20.639, -295]
  MoveL 3546 to (58.38, 27.56, -259.58) mm, rotated rx 105.8 ry 33.04 rz -145.95 deg; joints [-10.089, -24.714, 96.605, 141.211, 84.775, 20.598, -295]
  MoveL 3547 to (58.37, 27.98, -259.57) mm, rotated rx 105.8 ry 33.04 rz -145.95 deg; joints [-10.088, -24.732, 96.603, 141.211, 84.758, 20.611, -295]
  MoveC 3548 to (59.7, 31.27, -259.57) mm, rotated rx 105.8 ry 33.04 rz -145.95 deg; joints [-10.078, -24.802, 96.443, 141.207, 84.578, 20.752, -295] to (61.3, 34.45, -259.57) mm, rotated rx 105.8 ry 33.04 rz -145.95 deg; joints [-10.067, -24.851, 96.257, 141.203, 84.392, 20.898, -295]
  MoveL 3549 to (61.3, 34.45, -259.57) mm, rotated rx 105.8 ry 33.04 rz -145.95 deg; joints [-10.067, -24.851, 96.257, 141.203, 84.392, 20.898, -295]
  MoveL 3550 to (61.5, 34.87, -259.55) mm, rotated rx 105.8 ry 33.04 rz -145.95 deg; joints [-10.065, -24.858, 96.234, 141.204, 84.368, 20.917, -295]
  MoveL 3551 to (61.66, 35.26, -259.5) mm, rotated rx 105.8 ry 33.04 rz -145.95 deg; joints [-10.062, -24.866, 96.215, 141.205, 84.346, 20.933, -295]
  MoveL 3552 to (61.81, 35.64, -259.44) mm, rotated rx 105.8 ry 33.04 rz -145.95 deg; joints [-10.058, -24.874, 96.197, 141.207, 84.326, 20.948, -295]
  MoveL 3553 to (61.98, 36.04, -259.39) mm, rotated rx 105.8 ry 33.04 rz -145.95 deg; joints [-10.055, -24.882, 96.177, 141.208, 84.303, 20.965, -295]
  MoveL 3554 to (62.18, 36.47, -259.36) mm, rotated rx 105.8 ry 33.04 rz -145.95 deg; joints [-10.053, -24.89, 96.153, 141.208, 84.278, 20.984, -295]
  MoveL 3555 to (62.41, 36.94, -259.35) mm, rotated rx 105.8 ry 33.04 rz -145.95 deg; joints [-10.051, -24.897, 96.127, 141.208, 84.251, 21.005, -295]
  MoveL 3556 to (62.87, 37.88, -259.35) mm, rotated rx 105.8 ry 33.04 rz -145.95 deg; joints [-10.048, -24.912, 96.072, 141.207, 84.197, 21.048, -295]
  MoveL 3557 to (63.58, 39.15, -259.44) mm, rotated rx 105.8 ry 33.04 rz -145.95 deg; joints [-10.047, -24.928, 95.99, 141.202, 84.12, 21.109, -295]
  MoveL 3558 to (64.26, 40.14, -259.71) mm, rotated rx 105.8 ry 33.04 rz -145.95 deg; joints [-10.053, -24.931, 95.91, 141.19, 84.056, 21.164, -295]
  MoveL 3559 to (64.93, 40.84, -260.17) mm, rotated rx 105.8 ry 33.04 rz -145.95 deg; joints [-10.067, -24.924, 95.833, 141.172, 84.005, 21.211, -295]
  MoveL 3560 to (65.58, 41.24, -260.81) mm, rotated rx 105.8 ry 33.04 rz -145.95 deg; joints [-10.088, -24.904, 95.759, 141.148, 83.967, 21.251, -295]
  MoveL 3561 to (66.22, 41.37, -261.63) mm, rotated rx 105.8 ry 33.04 rz -145.95 deg; joints [-10.116, -24.873, 95.687, 141.118, 83.941, 21.284, -295]
  MoveL 3562 to (66.84, 41.2, -262.64) mm, rotated rx 105.8 ry 33.04 rz -145.95 deg; joints [-10.152, -24.831, 95.618, 141.081, 83.928, 21.31, -295]
  MoveL 3563 to (68.03, 40, -265.2) mm, rotated rx 105.8 ry 33.04 rz -145.95 deg; joints [-10.246, -24.711, 95.488, 140.989, 83.939, 21.34, -295]
  MoveL 3564 to (68.83, 38.11, -267.76) mm, rotated rx 105.8 ry 33.04 rz -145.95 deg; joints [-10.342, -24.583, 95.402, 140.899, 83.992, 21.338, -295]
  MoveL 3565 to (68.96, 37.08, -268.76) mm, rotated rx 105.8 ry 33.04 rz -145.95 deg; joints [-10.381, -24.53, 95.389, 140.863, 84.031, 21.323, -295]
  MoveL 3566 to (68.91, 35.99, -269.59) mm, rotated rx 105.8 ry 33.04 rz -145.95 deg; joints [-10.414, -24.486, 95.397, 140.835, 84.078, 21.299, -295]
  MoveL 3567 to (68.68, 34.85, -270.23) mm, rotated rx 105.8 ry 33.04 rz -145.95 deg; joints [-10.441, -24.449, 95.424, 140.813, 84.133, 21.265, -295]
  MoveL 3568 to (68.27, 33.66, -270.68) mm, rotated rx 105.8 ry 33.04 rz -145.95 deg; joints [-10.461, -24.42, 95.471, 140.798, 84.196, 21.221, -295]
  MoveL 3569 to (66.91, 31.1, -271.05) mm, rotated rx 105.8 ry 33.04 rz -145.95 deg; joints [-10.484, -24.384, 95.625, 140.788, 84.349, 21.106, -295]
  MoveL 3570 to (66.34, 30.22, -271.05) mm, rotated rx 105.8 ry 33.04 rz -145.95 deg; joints [-10.488, -24.377, 95.689, 140.789, 84.404, 21.062, -295]
  MoveL 3571 to (66.06, 29.78, -271.06) mm, rotated rx 105.8 ry 33.04 rz -145.95 deg; joints [-10.49, -24.373, 95.721, 140.789, 84.432, 21.04, -295]
  MoveL 3572 to (65.81, 29.37, -271.08) mm, rotated rx 105.8 ry 33.04 rz -145.95 deg; joints [-10.493, -24.369, 95.749, 140.788, 84.457, 21.021, -295]
  MoveL 3573 to (65.6, 29, -271.13) mm, rotated rx 105.8 ry 33.04 rz -145.95 deg; joints [-10.496, -24.364, 95.772, 140.787, 84.48, 21.004, -295]
  MoveL 3574 to (65.41, 28.65, -271.18) mm, rotated rx 105.8 ry 33.04 rz -145.95 deg; joints [-10.499, -24.359, 95.793, 140.785, 84.501, 20.988, -295]
  MoveL 3575 to (65.21, 28.28, -271.23) mm, rotated rx 105.8 ry 33.04 rz -145.95 deg; joints [-10.502, -24.354, 95.816, 140.784, 84.523, 20.971, -295]
  MoveL 3576 to (64.96, 27.88, -271.25) mm, rotated rx 105.8 ry 33.04 rz -145.95 deg; joints [-10.505, -24.35, 95.844, 140.783, 84.548, 20.952, -295]
  MoveL 3577 to (64.7, 27.46, -271.26) mm, rotated rx 105.8 ry 33.04 rz -145.95 deg; joints [-10.507, -24.347, 95.874, 140.783, 84.574, 20.931, -295]
  MoveL 3578 to (64.4, 26.99, -271.25) mm, rotated rx 105.8 ry 33.04 rz -145.95 deg; joints [-10.508, -24.343, 95.908, 140.784, 84.604, 20.907, -295]
  MoveL 3579 to (64.11, 26.55, -271.26) mm, rotated rx 105.8 ry 33.04 rz -145.95 deg; joints [-10.511, -24.339, 95.939, 140.784, 84.632, 20.885, -295]
  MoveL 3580 to (63.85, 26.13, -271.28) mm, rotated rx 105.8 ry 33.04 rz -145.95 deg; joints [-10.513, -24.335, 95.968, 140.784, 84.658, 20.865, -295]
  MoveL 3581 to (63.61, 25.72, -271.33) mm, rotated rx 105.8 ry 33.04 rz -145.95 deg; joints [-10.517, -24.33, 95.995, 140.782, 84.683, 20.845, -295]
  MoveL 3582 to (63.37, 25.27, -271.41) mm, rotated rx 105.8 ry 33.04 rz -145.95 deg; joints [-10.521, -24.324, 96.022, 140.78, 84.709, 20.826, -295]
  MoveL 3583 to (63.08, 24.74, -271.47) mm, rotated rx 105.8 ry 33.04 rz -145.95 deg; joints [-10.525, -24.317, 96.055, 140.778, 84.741, 20.801, -295]
  MoveL 3584 to (62.78, 24.26, -271.49) mm, rotated rx 105.8 ry 33.04 rz -145.95 deg; joints [-10.528, -24.312, 96.088, 140.777, 84.771, 20.778, -295]
  MoveL 3585 to (62.5, 23.81, -271.49) mm, rotated rx 105.8 ry 33.04 rz -145.95 deg; joints [-10.53, -24.308, 96.12, 140.778, 84.799, 20.755, -295]
  MoveL 3586 to (62.21, 23.37, -271.49) mm, rotated rx 105.8 ry 33.04 rz -145.95 deg; joints [-10.532, -24.304, 96.151, 140.778, 84.827, 20.733, -295]
  MoveL 3587 to (61.87, 22.81, -271.5) mm, rotated rx 105.8 ry 33.04 rz -145.95 deg; joints [-10.534, -24.298, 96.19, 140.778, 84.862, 20.706, -295]
  MoveL 3588 to (61.59, 22.3, -271.51) mm, rotated rx 105.8 ry 33.04 rz -145.95 deg; joints [-10.537, -24.291, 96.222, 140.778, 84.893, 20.682, -295]
  MoveL 3589 to (61.36, 21.85, -271.52) mm, rotated rx 105.8 ry 33.04 rz -145.95 deg; joints [-10.539, -24.284, 96.247, 140.778, 84.919, 20.661, -295]
  MoveL 3590 to (61.26, 21.52, -271.52) mm, rotated rx 105.8 ry 33.04 rz -145.95 deg; joints [-10.54, -24.275, 96.26, 140.778, 84.935, 20.648, -295]
  MoveL 3591 to (61.23, 21.25, -271.52) mm, rotated rx 105.8 ry 33.04 rz -145.95 deg; joints [-10.54, -24.266, 96.266, 140.778, 84.947, 20.638, -295]
  MoveL 3592 to (61.34, 22.18, -272.11) mm, rotated rx 105.8 ry 33.04 rz -145.95 deg; joints [-10.56, -24.298, 96.241, 140.756, 84.907, 20.679, -295]
  MoveL 3593 to (61.64, 20.88, -272.64) mm, rotated rx 105.8 ry 33.04 rz -145.95 deg; joints [-10.582, -24.225, 96.217, 140.738, 84.949, 20.654, -295]
  MoveL 3594 to (61.85, 19.33, -273.02) mm, rotated rx 105.8 ry 33.04 rz -145.95 deg; joints [-10.598, -24.147, 96.205, 140.725, 85.003, 20.616, -295]
  MoveL 3595 to (61.98, 17.49, -273.28) mm, rotated rx 105.8 ry 33.04 rz -145.95 deg; joints [-10.611, -24.061, 96.203, 140.717, 85.071, 20.565, -295]
  MoveL 3596 to (62.05, 15.44, -273.41) mm, rotated rx 105.8 ry 33.04 rz -145.95 deg; joints [-10.62, -23.969, 96.211, 140.715, 85.149, 20.504, -295]
  MoveL 3597 to (62.1, 13.33, -273.5) mm, rotated rx 105.8 ry 33.04 rz -145.95 deg; joints [-10.627, -23.876, 96.22, 140.713, 85.23, 20.441, -295]
  MoveL 3598 to (62.2, 9.07, -273.68) mm, rotated rx 105.8 ry 33.04 rz -145.95 deg; joints [-10.641, -23.687, 96.239, 140.709, 85.394, 20.312, -295]
  MoveL 3599 to (62.25, 6.94, -273.86) mm, rotated rx 105.8 ry 33.04 rz -145.95 deg; joints [-10.652, -23.592, 96.246, 140.704, 85.475, 20.249, -295]
  MoveL 3600 to (62.34, 2.67, -274.04) mm, rotated rx 105.8 ry 33.04 rz -145.95 deg; joints [-10.667, -23.403, 96.264, 140.7, 85.638, 20.121, -295]
  MoveL 3601 to (62.39, 0.54, -274.22) mm, rotated rx 105.8 ry 33.04 rz -145.95 deg; joints [-10.678, -23.307, 96.271, 140.694, 85.72, 20.058, -295]
  MoveL 3602 to (62.43, -1.6, -274.31) mm, rotated rx 105.8 ry 33.04 rz -145.95 deg; joints [-10.685, -23.212, 96.279, 140.692, 85.801, 19.995, -295]
  MoveL 3603 to (62.44, -3.57, -274.52) mm, rotated rx 105.8 ry 33.04 rz -145.95 deg; joints [-10.697, -23.125, 96.288, 140.685, 85.877, 19.936, -295]
  MoveL 3604 to (62.48, -5.93, -274.67) mm, rotated rx 105.8 ry 33.04 rz -145.95 deg; joints [-10.707, -23.019, 96.296, 140.68, 85.967, 19.867, -295]
  MoveL 3605 to (62.53, -8.49, -274.79) mm, rotated rx 105.8 ry 33.04 rz -145.95 deg; joints [-10.716, -22.904, 96.304, 140.677, 86.064, 19.79, -295]
  MoveL 3606 to (62.57, -10.63, -274.79) mm, rotated rx 105.8 ry 33.04 rz -145.95 deg; joints [-10.72, -22.809, 96.312, 140.677, 86.145, 19.726, -295]
  MoveL 3607 to (62.6, -12.66, -274.86) mm, rotated rx 105.8 ry 33.04 rz -145.95 deg; joints [-10.727, -22.718, 96.319, 140.675, 86.222, 19.665, -295]
  MoveL 3608 to (62.61, -14.49, -275.04) mm, rotated rx 105.8 ry 33.04 rz -145.95 deg; joints [-10.737, -22.636, 96.325, 140.669, 86.292, 19.611, -295]
  MoveL 3609 to (62.61, -16.36, -275.25) mm, rotated rx 105.8 ry 33.04 rz -145.95 deg; joints [-10.749, -22.553, 96.333, 140.661, 86.364, 19.556, -295]
  MoveL 3610 to (62.64, -18.72, -275.38) mm, rotated rx 105.8 ry 33.04 rz -145.95 deg; joints [-10.759, -22.447, 96.34, 140.656, 86.453, 19.486, -295]
  MoveL 3611 to (62.67, -21.3, -275.49) mm, rotated rx 105.8 ry 33.04 rz -145.95 deg; joints [-10.768, -22.33, 96.347, 140.652, 86.55, 19.41, -295]
  MoveL 3612 to (62.75, -25.56, -275.49) mm, rotated rx 105.8 ry 33.04 rz -145.95 deg; joints [-10.776, -22.137, 96.358, 140.652, 86.71, 19.282, -295]
  MoveL 3613 to (62.52, -25.78, -276.19) mm, rotated rx 105.8 ry 33.04 rz -145.95 deg; joints [-10.804, -22.137, 96.375, 140.625, 86.727, 19.277, -295]
  MoveL 3614 to (62.39, -25.49, -276.53) mm, rotated rx 105.8 ry 33.04 rz -145.95 deg; joints [-10.817, -22.155, 96.383, 140.612, 86.722, 19.286, -295]
  MoveL 3615 to (62.37, -25.49, -276.75) mm, rotated rx 105.8 ry 33.04 rz -145.95 deg; joints [-10.825, -22.156, 96.382, 140.604, 86.722, 19.288, -295]
  MoveL 3616 to (62.46, -25.74, -276.86) mm, rotated rx 105.8 ry 33.04 rz -145.95 deg; joints [-10.829, -22.14, 96.373, 140.6, 86.729, 19.285, -295]
  MoveL 3617 to (62.67, -26.14, -276.89) mm, rotated rx 105.8 ry 33.04 rz -145.95 deg; joints [-10.831, -22.111, 96.354, 140.599, 86.736, 19.279, -295]
  MoveL 3618 to (62.91, -26.55, -276.92) mm, rotated rx 105.8 ry 33.04 rz -145.95 deg; joints [-10.831, -22.081, 96.331, 140.599, 86.742, 19.274, -295]
  MoveL 3619 to (63.14, -26.92, -276.96) mm, rotated rx 105.8 ry 33.04 rz -145.95 deg; joints [-10.833, -22.053, 96.31, 140.597, 86.748, 19.27, -295]
  MoveL 3620 to (63.34, -27.27, -277.03) mm, rotated rx 105.8 ry 33.04 rz -145.95 deg; joints [-10.836, -22.027, 96.291, 140.595, 86.753, 19.267, -295]
  MoveL 3621 to (63.55, -27.62, -277.09) mm, rotated rx 105.8 ry 33.04 rz -145.95 deg; joints [-10.838, -22, 96.271, 140.593, 86.759, 19.263, -295]
  MoveL 3622 to (63.79, -27.99, -277.13) mm, rotated rx 105.8 ry 33.04 rz -145.95 deg; joints [-10.839, -21.971, 96.248, 140.592, 86.764, 19.259, -295]
  MoveL 3623 to (64.08, -28.43, -277.15) mm, rotated rx 105.8 ry 33.04 rz -145.95 deg; joints [-10.84, -21.937, 96.221, 140.592, 86.769, 19.255, -295]
  MoveL 3624 to (64.36, -28.88, -277.22) mm, rotated rx 105.8 ry 33.04 rz -145.95 deg; joints [-10.842, -21.903, 96.195, 140.59, 86.776, 19.25, -295]
  MoveL 3625 to (64.64, -29.32, -277.25) mm, rotated rx 105.8 ry 33.04 rz -145.95 deg; joints [-10.843, -21.869, 96.168, 140.589, 86.782, 19.246, -295]
  MoveL 3626 to (64.94, -29.75, -277.25) mm, rotated rx 105.8 ry 33.04 rz -145.95 deg; joints [-10.843, -21.835, 96.14, 140.589, 86.786, 19.242, -295]
  MoveL 3627 to (65.24, -30.18, -277.25) mm, rotated rx 105.8 ry 33.04 rz -145.95 deg; joints [-10.843, -21.8, 96.112, 140.59, 86.791, 19.238, -295]
  MoveL 3628 to (65.64, -30.73, -277.22) mm, rotated rx 105.8 ry 33.04 rz -145.95 deg; joints [-10.841, -21.755, 96.074, 140.591, 86.797, 19.233, -295]
  MoveL 3629 to (66.04, -31.27, -277.19) mm, rotated rx 105.8 ry 33.04 rz -145.95 deg; joints [-10.84, -21.711, 96.037, 140.593, 86.802, 19.228, -295]
  MoveL 3630 to (66.38, -31.76, -277.18) mm, rotated rx 105.8 ry 33.04 rz -145.95 deg; joints [-10.839, -21.672, 96.005, 140.594, 86.807, 19.224, -295]
  MoveL 3631 to (66.63, -32.16, -277.22) mm, rotated rx 105.8 ry 33.04 rz -145.95 deg; joints [-10.84, -21.641, 95.981, 140.593, 86.812, 19.22, -295]
  MoveL 3632 to (66.84, -32.51, -277.28) mm, rotated rx 105.8 ry 33.04 rz -145.95 deg; joints [-10.843, -21.615, 95.961, 140.591, 86.818, 19.216, -295]
  MoveL 3633 to (67.05, -32.86, -277.34) mm, rotated rx 105.8 ry 33.04 rz -145.95 deg; joints [-10.845, -21.588, 95.94, 140.589, 86.823, 19.213, -295]
  MoveL 3634 to (67.29, -33.23, -277.37) mm, rotated rx 105.8 ry 33.04 rz -145.95 deg; joints [-10.846, -21.559, 95.918, 140.588, 86.828, 19.209, -295]
  MoveL 3635 to (68.19, -34.52, -277.37) mm, rotated rx 105.8 ry 33.04 rz -145.95 deg; joints [-10.845, -21.456, 95.833, 140.59, 86.842, 19.197, -295]
  MoveL 3636 to (69.65, -37.02, -277.75) mm, rotated rx 105.8 ry 33.04 rz -145.95 deg; joints [-10.859, -21.27, 95.692, 140.578, 86.879, 19.171, -295]
  MoveL 3637 to (70.11, -38.18, -278.22) mm, rotated rx 105.8 ry 33.04 rz -145.95 deg; joints [-10.877, -21.193, 95.645, 140.561, 86.905, 19.156, -295]
  MoveL 3638 to (70.4, -39.29, -278.88) mm, rotated rx 105.8 ry 33.04 rz -145.95 deg; joints [-10.903, -21.127, 95.613, 140.537, 86.936, 19.14, -295]
  MoveL 3639 to (70.51, -40.34, -279.72) mm, rotated rx 105.8 ry 33.04 rz -145.95 deg; joints [-10.937, -21.072, 95.597, 140.505, 86.972, 19.122, -295]
  MoveL 3640 to (70.44, -41.34, -280.76) mm, rotated rx 105.8 ry 33.04 rz -145.95 deg; joints [-10.979, -21.028, 95.596, 140.466, 87.012, 19.103, -295]
  MoveL 3641 to (69.77, -43.17, -283.4) mm, rotated rx 105.8 ry 33.04 rz -145.95 deg; joints [-11.085, -20.973, 95.641, 140.365, 87.107, 19.061, -295]
  MoveL 3642 to (68.68, -44.33, -286.03) mm, rotated rx 105.8 ry 33.04 rz -145.95 deg; joints [-11.192, -20.968, 95.725, 140.264, 87.194, 19.026, -295]
  MoveL 3643 to (68.09, -44.48, -287.07) mm, rotated rx 105.8 ry 33.04 rz -145.95 deg; joints [-11.234, -20.988, 95.774, 140.224, 87.223, 19.016, -295]
  MoveL 3644 to (67.46, -44.36, -287.92) mm, rotated rx 105.8 ry 33.04 rz -145.95 deg; joints [-11.268, -21.023, 95.827, 140.191, 87.243, 19.011, -295]
  MoveL 3645 to (66.81, -43.95, -288.58) mm, rotated rx 105.8 ry 33.04 rz -145.95 deg; joints [-11.295, -21.073, 95.884, 140.165, 87.253, 19.012, -295]
  MoveL 3646 to (66.12, -43.27, -289.05) mm, rotated rx 105.8 ry 33.04 rz -145.95 deg; joints [-11.314, -21.137, 95.946, 140.147, 87.254, 19.017, -295]
  MoveL 3647 to (65.39, -42.3, -289.33) mm, rotated rx 105.8 ry 33.04 rz -145.95 deg; joints [-11.326, -21.216, 96.012, 140.135, 87.246, 19.028, -295]
  MoveL 3648 to (64.64, -41.05, -289.42) mm, rotated rx 105.8 ry 33.04 rz -145.95 deg; joints [-11.33, -21.31, 96.082, 140.13, 87.229, 19.044, -295]
  MoveL 3649 to (64.38, -40.6, -289.42) mm, rotated rx 105.8 ry 33.04 rz -145.95 deg; joints [-11.33, -21.343, 96.106, 140.13, 87.222, 19.05, -295]
  MoveL 3650 to (64.17, -40.18, -289.4) mm, rotated rx 105.8 ry 33.04 rz -145.95 deg; joints [-11.329, -21.373, 96.127, 140.13, 87.215, 19.055, -295]
  MoveL 3651 to (63.99, -39.82, -289.36) mm, rotated rx 105.8 ry 33.04 rz -145.95 deg; joints [-11.327, -21.398, 96.143, 140.132, 87.208, 19.061, -295]
  MoveL 3652 to (63.83, -39.46, -289.3) mm, rotated rx 105.8 ry 33.04 rz -145.95 deg; joints [-11.325, -21.423, 96.159, 140.134, 87.201, 19.066, -295]
  MoveL 3653 to (63.64, -39.07, -289.26) mm, rotated rx 105.8 ry 33.04 rz -145.95 deg; joints [-11.323, -21.45, 96.177, 140.135, 87.193, 19.071, -295]
  MoveL 3654 to (63.41, -38.64, -289.23) mm, rotated rx 105.8 ry 33.04 rz -145.95 deg; joints [-11.322, -21.481, 96.199, 140.136, 87.186, 19.077, -295]
  MoveL 3655 to (63.16, -38.18, -289.23) mm, rotated rx 105.8 ry 33.04 rz -145.95 deg; joints [-11.322, -21.514, 96.222, 140.136, 87.178, 19.083, -295]
  MoveL 3656 to (62.94, -37.77, -289.21) mm, rotated rx 105.8 ry 33.04 rz -145.95 deg; joints [-11.322, -21.544, 96.243, 140.136, 87.171, 19.089, -295]
  MoveL 3657 to (62.76, -37.41, -289.16) mm, rotated rx 105.8 ry 33.04 rz -145.95 deg; joints [-11.319, -21.569, 96.261, 140.138, 87.165, 19.094, -295]
  MoveL 3658 to (62.59, -37.06, -289.1) mm, rotated rx 105.8 ry 33.04 rz -145.95 deg; joints [-11.317, -21.594, 96.277, 140.14, 87.158, 19.098, -295]
  MoveL 3659 to (62.39, -36.67, -289.05) mm, rotated rx 105.8 ry 33.04 rz -145.95 deg; joints [-11.315, -21.621, 96.296, 140.141, 87.151, 19.104, -295]
  MoveL 3660 to (62.16, -36.24, -289.03) mm, rotated rx 105.8 ry 33.04 rz -145.95 deg; joints [-11.314, -21.652, 96.317, 140.142, 87.144, 19.109, -295]
  MoveL 3661 to (61.91, -35.78, -289.03) mm, rotated rx 105.8 ry 33.04 rz -145.95 deg; joints [-11.314, -21.686, 96.341, 140.142, 87.137, 19.116, -295]
  MoveL 3662 to (61.49, -34.89, -289.01) mm, rotated rx 105.8 ry 33.04 rz -145.95 deg; joints [-11.313, -21.747, 96.379, 140.142, 87.119, 19.13, -295]
  MoveC 3663 to (60.95, -33.62, -289.01) mm, rotated rx 105.8 ry 33.04 rz -145.95 deg; joints [-11.313, -21.831, 96.429, 140.141, 87.092, 19.153, -295] to (60.25, -32.43, -289.01) mm, rotated rx 105.8 ry 33.04 rz -145.95 deg; joints [-11.313, -21.92, 96.493, 140.14, 87.073, 19.168, -295]
  MoveL 3664 to (60.25, -32.43, -289) mm, rotated rx 105.8 ry 33.04 rz -145.95 deg; joints [-11.313, -21.92, 96.493, 140.141, 87.073, 19.168, -295]
  MoveL 3665 to (59.97, -31.83, -288.98) mm, rotated rx 105.8 ry 33.04 rz -145.95 deg; joints [-11.312, -21.961, 96.52, 140.141, 87.062, 19.177, -295]
  MoveL 3666 to (59.78, -31.29, -288.96) mm, rotated rx 105.8 ry 33.04 rz -145.95 deg; joints [-11.311, -21.995, 96.537, 140.142, 87.049, 19.188, -295]
  MoveL 3667 to (59.74, -30.99, -288.86) mm, rotated rx 105.8 ry 33.04 rz -145.95 deg; joints [-11.306, -22.011, 96.54, 140.145, 87.039, 19.195, -295]
  MoveL 3668 to (59.8, -31.02, -288.66) mm, rotated rx 105.8 ry 33.04 rz -145.95 deg; joints [-11.299, -22.007, 96.537, 140.153, 87.038, 19.193, -295]
  MoveL 3669 to (59.93, -31.42, -288.35) mm, rotated rx 105.8 ry 33.04 rz -145.95 deg; joints [-11.287, -21.983, 96.528, 140.164, 87.048, 19.181, -295]
  MoveL 3670 to (60.3, -31.52, -287.73) mm, rotated rx 105.8 ry 33.04 rz -145.95 deg; joints [-11.263, -21.961, 96.499, 140.188, 87.037, 19.181, -295]
  MoveL 3671 to (60.37, -29.49, -287.72) mm, rotated rx 105.8 ry 33.04 rz -145.95 deg; joints [-11.258, -22.049, 96.485, 140.19, 86.958, 19.245, -295]
  MoveL 3672 to (60.52, -27.35, -287.67) mm, rotated rx 105.8 ry 33.04 rz -145.95 deg; joints [-11.25, -22.137, 96.462, 140.193, 86.872, 19.315, -295]
  MoveL 3673 to (60.72, -25.09, -287.54) mm, rotated rx 105.8 ry 33.04 rz -145.95 deg; joints [-11.24, -22.228, 96.434, 140.199, 86.778, 19.389, -295]
  MoveL 3674 to (60.92, -22.86, -287.44) mm, rotated rx 105.8 ry 33.04 rz -145.95 deg; joints [-11.231, -22.318, 96.406, 140.203, 86.686, 19.462, -295]
  MoveL 3675 to (61.12, -20.72, -287.27) mm, rotated rx 105.8 ry 33.04 rz -145.95 deg; joints [-11.219, -22.403, 96.378, 140.211, 86.598, 19.532, -295]
  MoveL 3676 to (61.3, -18.78, -287.12) mm, rotated rx 105.8 ry 33.04 rz -145.95 deg; joints [-11.209, -22.48, 96.353, 140.217, 86.517, 19.596, -295]
  MoveL 3677 to (61.48, -16.72, -287.07) mm, rotated rx 105.8 ry 33.04 rz -145.95 deg; joints [-11.202, -22.562, 96.326, 140.219, 86.432, 19.664, -295]
  MoveL 3678 to (61.67, -14.57, -287) mm, rotated rx 105.8 ry 33.04 rz -145.95 deg; joints [-11.194, -22.648, 96.298, 140.222, 86.343, 19.735, -295]
  MoveL 3679 to (61.87, -12.23, -286.85) mm, rotated rx 105.8 ry 33.04 rz -145.95 deg; joints [-11.182, -22.741, 96.267, 140.228, 86.246, 19.812, -295]
  MoveL 3680 to (62.04, -10.36, -286.73) mm, rotated rx 105.8 ry 33.04 rz -145.95 deg; joints [-11.174, -22.815, 96.242, 140.233, 86.168, 19.874, -295]
  MoveL 3681 to (62.24, -7.98, -286.52) mm, rotated rx 105.8 ry 33.04 rz -145.95 deg; joints [-11.16, -22.91, 96.212, 140.241, 86.07, 19.951, -295]
  MoveL 3682 to (62.39, -6.1, -286.41) mm, rotated rx 105.8 ry 33.04 rz -145.95 deg; joints [-11.151, -22.984, 96.187, 140.245, 85.992, 20.012, -295]
  MoveL 3683 to (62.57, -3.98, -286.24) mm, rotated rx 105.8 ry 33.04 rz -145.95 deg; joints [-11.14, -23.068, 96.159, 140.251, 85.904, 20.082, -295]
  MoveL 3684 to (62.76, -1.6, -286.19) mm, rotated rx 105.8 ry 33.04 rz -145.95 deg; joints [-11.132, -23.162, 96.126, 140.252, 85.805, 20.161, -295]
  MoveL 3685 to (62.91, 0.28, -286.08) mm, rotated rx 105.8 ry 33.04 rz -145.95 deg; joints [-11.123, -23.236, 96.101, 140.256, 85.727, 20.223, -295]
  MoveL 3686 to (63.08, 2.4, -285.92) mm, rotated rx 105.8 ry 33.04 rz -145.95 deg; joints [-11.112, -23.32, 96.073, 140.262, 85.639, 20.292, -295]
  MoveL 3687 to (63.27, 4.78, -285.87) mm, rotated rx 105.8 ry 33.04 rz -145.95 deg; joints [-11.105, -23.413, 96.039, 140.263, 85.54, 20.372, -295]
  MoveL 3688 to (63.42, 6.66, -285.75) mm, rotated rx 105.8 ry 33.04 rz -145.95 deg; joints [-11.096, -23.486, 96.013, 140.266, 85.462, 20.433, -295]
  MoveL 3689 to (63.59, 8.87, -285.65) mm, rotated rx 105.8 ry 33.04 rz -145.95 deg; joints [-11.087, -23.573, 95.982, 140.269, 85.369, 20.507, -295]
  MoveL 3690 to (63.76, 11.09, -285.58) mm, rotated rx 105.8 ry 33.04 rz -145.95 deg; joints [-11.079, -23.659, 95.95, 140.27, 85.277, 20.581, -295]
  MoveL 3691 to (63.87, 12.97, -285.4) mm, rotated rx 105.8 ry 33.04 rz -145.95 deg; joints [-11.068, -23.734, 95.927, 140.276, 85.199, 20.641, -295]
  MoveL 3692 to (63.95, 14.7, -285.15) mm, rotated rx 105.8 ry 33.04 rz -145.95 deg; joints [-11.055, -23.805, 95.909, 140.284, 85.129, 20.695, -295]
  MoveL 3693 to (64, 16.32, -284.8) mm, rotated rx 105.8 ry 33.04 rz -145.95 deg; joints [-11.038, -23.873, 95.897, 140.296, 85.063, 20.742, -295]
  MoveL 3694 to (63.46, 14.92, -284.11) mm, rotated rx 105.8 ry 33.04 rz -145.95 deg; joints [-11.017, -23.843, 95.968, 140.321, 85.137, 20.673, -295]
  MoveL 3695 to (63.52, 15.14, -284.1) mm, rotated rx 105.8 ry 33.04 rz -145.95 deg; joints [-11.017, -23.85, 95.96, 140.321, 85.126, 20.681, -295]
  MoveL 3696 to (63.63, 15.41, -284.09) mm, rotated rx 105.8 ry 33.04 rz -145.95 deg; joints [-11.015, -23.855, 95.947, 140.322, 85.111, 20.693, -295]
  MoveL 3697 to (63.87, 15.8, -284.06) mm, rotated rx 105.8 ry 33.04 rz -145.95 deg; joints [-11.012, -23.859, 95.92, 140.323, 85.087, 20.712, -295]
  MoveL 3698 to (64.18, 16.25, -284.02) mm, rotated rx 105.8 ry 33.04 rz -145.95 deg; joints [-11.009, -23.863, 95.888, 140.324, 85.058, 20.735, -295]
  MoveL 3699 to (64.54, 16.74, -283.98) mm, rotated rx 105.8 ry 33.04 rz -145.95 deg; joints [-11.005, -23.865, 95.848, 140.326, 85.026, 20.76, -295]
  MoveL 3700 to (66.17, 18.79, -283.98) mm, rotated rx 105.8 ry 33.04 rz -145.95 deg; joints [-10.994, -23.866, 95.67, 140.326, 84.886, 20.873, -295]
  MoveL 3701 to (66.54, 19.28, -283.95) mm, rotated rx 105.8 ry 33.04 rz -145.95 deg; joints [-10.991, -23.868, 95.631, 140.327, 84.853, 20.898, -295]
  MoveL 3702 to (66.94, 19.83, -283.89) mm, rotated rx 105.8 ry 33.04 rz -145.95 deg; joints [-10.986, -23.87, 95.587, 140.329, 84.817, 20.927, -295]
  MoveL 3703 to (67.32, 20.33, -283.86) mm, rotated rx 105.8 ry 33.04 rz -145.95 deg; joints [-10.983, -23.872, 95.546, 140.33, 84.783, 20.953, -295]
  MoveL 3704 to (67.65, 20.74, -283.86) mm, rotated rx 105.8 ry 33.04 rz -145.95 deg; joints [-10.981, -23.872, 95.51, 140.33, 84.755, 20.976, -295]
  MoveL 3705 to (67.95, 21.13, -283.85) mm, rotated rx 105.8 ry 33.04 rz -145.95 deg; joints [-10.978, -23.872, 95.476, 140.33, 84.729, 20.997, -295]
  MoveL 3706 to (68.28, 21.53, -283.85) mm, rotated rx 105.8 ry 33.04 rz -145.95 deg; joints [-10.976, -23.872, 95.441, 140.33, 84.701, 21.019, -295]
  MoveL 3707 to (68.6, 21.94, -283.85) mm, rotated rx 105.8 ry 33.04 rz -145.95 deg; joints [-10.974, -23.872, 95.406, 140.33, 84.673, 21.041, -295]
  MoveL 3708 to (68.89, 22.32, -283.82) mm, rotated rx 105.8 ry 33.04 rz -145.95 deg; joints [-10.971, -23.873, 95.373, 140.331, 84.647, 21.062, -295]
  MoveL 3709 to (69.17, 22.7, -283.77) mm, rotated rx 105.8 ry 33.04 rz -145.95 deg; joints [-10.968, -23.874, 95.344, 140.332, 84.623, 21.081, -295]
  MoveL 3710 to (69.47, 23.09, -283.75) mm, rotated rx 105.8 ry 33.04 rz -145.95 deg; joints [-10.965, -23.875, 95.311, 140.333, 84.596, 21.102, -295]
  MoveL 3711 to (69.8, 23.51, -283.75) mm, rotated rx 105.8 ry 33.04 rz -145.95 deg; joints [-10.963, -23.875, 95.274, 140.333, 84.568, 21.124, -295]
  MoveL 3712 to (70.46, 24.32, -283.75) mm, rotated rx 105.8 ry 33.04 rz -145.95 deg; joints [-10.959, -23.875, 95.202, 140.332, 84.512, 21.169, -295]
  Set speed (1000.0 mm/s)
  MoveL 3713 to (88.16, 36.72, -283.75) mm, rotated rx 105.8 ry 33.04 rz -145.95 deg; joints [-10.87, -23.44, 93.312, 140.32, 83.373, 22.081, -295]
  Print: /'Flow1'
  Set speed (1000.0 mm/s)
  MoveL 3714 to (-79.06, 86.72, -80.22) mm, rotated rx 42.04 ry 15.1 rz -114.75 deg; joints [-11.881, -44.556, 105.513, 149.142, 46.632, -28.661, -355]
  Set speed (1000.0 mm/s)
  MoveL 3715 to (-75.15, 42.01, -80.22) mm, rotated rx 42.04 ry 15.1 rz -114.75 deg; joints [-12.109, -45.867, 109.411, 150.046, 48.916, -30.305, -355]
  Set speed (100.0 mm/s)
  MoveL 3716 to (-68.81, -30.47, -80.22) mm, rotated rx 42.04 ry 15.1 rz -114.75 deg; joints [-12.508, -47.756, 115.477, 151.236, 52.637, -32.762, -355]
  MoveL 3717 to (-69.1, -30.91, -80.22) mm, rotated rx 42.04 ry 15.1 rz -114.75 deg; joints [-12.511, -47.788, 115.518, 151.237, 52.647, -32.767, -355]
  MoveL 3718 to (-69.4, -31.48, -80.12) mm, rotated rx 42.04 ry 15.1 rz -114.75 deg; joints [-12.51, -47.824, 115.571, 151.244, 52.661, -32.777, -355]
  MoveL 3719 to (-69.7, -31.99, -80.06) mm, rotated rx 42.04 ry 15.1 rz -114.75 deg; joints [-12.511, -47.858, 115.619, 151.248, 52.674, -32.786, -355]
  MoveL 3720 to (-70, -32.47, -80.04) mm, rotated rx 42.04 ry 15.1 rz -114.75 deg; joints [-12.513, -47.891, 115.664, 151.25, 52.685, -32.792, -355]
  MoveL 3721 to (-72, -35.54, -80.04) mm, rotated rx 42.04 ry 15.1 rz -114.75 deg; joints [-12.532, -48.109, 115.952, 151.254, 52.75, -32.827, -355]
  MoveL 3722 to (-72.84, -36.72, -80.13) mm, rotated rx 42.04 ry 15.1 rz -114.75 deg; joints [-12.542, -48.197, 116.063, 151.249, 52.771, -32.836, -355]
  MoveL 3723 to (-73.64, -37.61, -80.4) mm, rotated rx 42.04 ry 15.1 rz -114.75 deg; joints [-12.559, -48.272, 116.146, 151.233, 52.781, -32.834, -355]
  MoveL 3724 to (-74.38, -38.19, -80.84) mm, rotated rx 42.04 ry 15.1 rz -114.75 deg; joints [-12.581, -48.334, 116.201, 151.204, 52.779, -32.82, -355]
  MoveL 3725 to (-74.73, -38.37, -81.13) mm, rotated rx 42.04 ry 15.1 rz -114.75 deg; joints [-12.594, -48.361, 116.218, 151.185, 52.774, -32.809, -355]
  MoveL 3726 to (-75.07, -38.48, -81.46) mm, rotated rx 42.04 ry 15.1 rz -114.75 deg; joints [-12.609, -48.384, 116.229, 151.163, 52.765, -32.795, -355]
  MoveL 3727 to (-75.72, -38.47, -82.26) mm, rotated rx 42.04 ry 15.1 rz -114.75 deg; joints [-12.642, -48.421, 116.229, 151.11, 52.739, -32.759, -355]
  MoveL 3728 to (-76.31, -38.17, -83.24) mm, rotated rx 42.04 ry 15.1 rz -114.75 deg; joints [-12.682, -48.445, 116.202, 151.045, 52.701, -32.712, -355]
  MoveL 3729 to (-77.36, -36.66, -85.72) mm, rotated rx 42.04 ry 15.1 rz -114.75 deg; joints [-12.777, -48.455, 116.064, 150.878, 52.589, -32.582, -355]
  MoveL 3730 to (-77.93, -34.52, -88.21) mm, rotated rx 42.04 ry 15.1 rz -114.75 deg; joints [-12.867, -48.415, 115.865, 150.712, 52.467, -32.446, -355]
  MoveL 3731 to (-77.76, -32.29, -89.98) mm, rotated rx 42.04 ry 15.1 rz -114.75 deg; joints [-12.927, -48.329, 115.655, 150.594, 52.371, -32.344, -355]
  MoveL 3732 to (-77.39, -31.15, -90.6) mm, rotated rx 42.04 ry 15.1 rz -114.75 deg; joints [-12.946, -48.269, 115.547, 150.554, 52.332, -32.306, -355]
  MoveL 3733 to (-76.84, -29.98, -91.05) mm, rotated rx 42.04 ry 15.1 rz -114.75 deg; joints [-12.957, -48.197, 115.435, 150.526, 52.3, -32.277, -355]
  MoveL 3734 to (-75.19, -27.58, -91.4) mm, rotated rx 42.04 ry 15.1 rz -114.75 deg; joints [-12.956, -48.019, 115.205, 150.507, 52.254, -32.244, -355]
  MoveL 3735 to (-73.18, -25.16, -91.41) mm, rotated rx 42.04 ry 15.1 rz -114.75 deg; joints [-12.941, -47.82, 114.97, 150.511, 52.22, -32.229, -355]
  MoveL 3736 to (-72.87, -24.77, -91.43) mm, rotated rx 42.04 ry 15.1 rz -114.75 deg; joints [-12.94, -47.789, 114.933, 150.51, 52.214, -32.225, -355]
  MoveL 3737 to (-72.6, -24.4, -91.47) mm, rotated rx 42.04 ry 15.1 rz -114.75 deg; joints [-12.939, -47.761, 114.897, 150.508, 52.208, -32.221, -355]
  MoveL 3738 to (-72.37, -24.06, -91.53) mm, rotated rx 42.04 ry 15.1 rz -114.75 deg; joints [-12.939, -47.735, 114.864, 150.505, 52.201, -32.216, -355]
  MoveL 3739 to (-72.11, -23.7, -91.58) mm, rotated rx 42.04 ry 15.1 rz -114.75 deg; joints [-12.939, -47.708, 114.829, 150.502, 52.194, -32.211, -355]
  MoveL 3740 to (-71.77, -23.27, -91.6) mm, rotated rx 42.04 ry 15.1 rz -114.75 deg; joints [-12.937, -47.674, 114.787, 150.501, 52.187, -32.207, -355]
  MoveL 3741 to (-71.37, -22.75, -91.64) mm, rotated rx 42.04 ry 15.1 rz -114.75 deg; joints [-12.936, -47.633, 114.737, 150.5, 52.179, -32.202, -355]
  MoveL 3742 to (-71.04, -22.3, -91.7) mm, rotated rx 42.04 ry 15.1 rz -114.75 deg; joints [-12.935, -47.599, 114.693, 150.497, 52.171, -32.197, -355]
  MoveL 3743 to (-70.79, -21.93, -91.77) mm, rotated rx 42.04 ry 15.1 rz -114.75 deg; joints [-12.936, -47.571, 114.657, 150.493, 52.163, -32.191, -355]
  MoveL 3744 to (-70.54, -21.58, -91.82) mm, rotated rx 42.04 ry 15.1 rz -114.75 deg; joints [-12.936, -47.545, 114.623, 150.49, 52.157, -32.186, -355]
  MoveL 3745 to (-70.24, -21.2, -91.84) mm, rotated rx 42.04 ry 15.1 rz -114.75 deg; joints [-12.934, -47.515, 114.586, 150.489, 52.151, -32.183, -355]
  MoveL 3746 to (-69.91, -20.8, -91.84) mm, rotated rx 42.04 ry 15.1 rz -114.75 deg; joints [-12.932, -47.482, 114.547, 150.49, 52.145, -32.18, -355]
  MoveL 3747 to (-69.56, -20.38, -91.85) mm, rotated rx 42.04 ry 15.1 rz -114.75 deg; joints [-12.929, -47.448, 114.506, 150.491, 52.139, -32.177, -355]
  MoveL 3748 to (-69.21, -19.93, -91.86) mm, rotated rx 42.04 ry 15.1 rz -114.75 deg; joints [-12.927, -47.412, 114.463, 150.49, 52.131, -32.173, -355]
  MoveL 3749 to (-68.81, -19.4, -91.89) mm, rotated rx 42.04 ry 15.1 rz -114.75 deg; joints [-12.925, -47.371, 114.412, 150.489, 52.122, -32.168, -355]
  MoveL 3750 to (-68.49, -18.91, -91.96) mm, rotated rx 42.04 ry 15.1 rz -114.75 deg; joints [-12.924, -47.335, 114.364, 150.485, 52.112, -32.16, -355]
  MoveL 3751 to (-68.26, -18.52, -92.06) mm, rotated rx 42.04 ry 15.1 rz -114.75 deg; joints [-12.926, -47.309, 114.326, 150.478, 52.102, -32.153, -355]
  MoveL 3752 to (-68.25, -18.52, -92.3) mm, rotated rx 42.04 ry 15.1 rz -114.75 deg; joints [-12.936, -47.307, 114.324, 150.466, 52.103, -32.148, -355]
  MoveL 3753 to (-68.39, -18.89, -92.65) mm, rotated rx 42.04 ry 15.1 rz -114.75 deg; joints [-12.953, -47.325, 114.353, 150.45, 52.115, -32.147, -355]
  MoveL 3754 to (-69.21, -19.13, -93.61) mm, rotated rx 42.04 ry 15.1 rz -114.75 deg; joints [-12.994, -47.379, 114.374, 150.389, 52.095, -32.109, -355]
  MoveL 3755 to (-68.99, -17.01, -93.61) mm, rotated rx 42.04 ry 15.1 rz -114.75 deg; joints [-12.981, -47.301, 114.192, 150.365, 52.003, -32.05, -355]
  MoveL 3756 to (-68.79, -14.72, -93.74) mm, rotated rx 42.04 ry 15.1 rz -114.75 deg; joints [-12.972, -47.219, 113.996, 150.33, 51.902, -31.982, -355]
  MoveL 3757 to (-68.58, -12.55, -93.8) mm, rotated rx 42.04 ry 15.1 rz -114.75 deg; joints [-12.961, -47.139, 113.809, 150.302, 51.807, -31.919, -355]
  MoveL 3758 to (-68.38, -10.44, -93.93) mm, rotated rx 42.04 ry 15.1 rz -114.75 deg; joints [-12.954, -47.062, 113.627, 150.27, 51.714, -31.856, -355]
  MoveL 3759 to (-68.18, -8.3, -94.09) mm, rotated rx 42.04 ry 15.1 rz -114.75 deg; joints [-12.947, -46.984, 113.442, 150.236, 51.62, -31.791, -355]
  MoveL 3760 to (-67.98, -6.19, -94.21) mm, rotated rx 42.04 ry 15.1 rz -114.75 deg; joints [-12.94, -46.906, 113.259, 150.203, 51.527, -31.728, -355]
  MoveL 3761 to (-67.78, -4.06, -94.42) mm, rotated rx 42.04 ry 15.1 rz -114.75 deg; joints [-12.935, -46.827, 113.073, 150.166, 51.433, -31.662, -355]
  MoveL 3762 to (-67.57, -1.94, -94.54) mm, rotated rx 42.04 ry 15.1 rz -114.75 deg; joints [-12.927, -46.748, 112.889, 150.134, 51.34, -31.599, -355]
  MoveL 3763 to (-67.36, 0.19, -94.59) mm, rotated rx 42.04 ry 15.1 rz -114.75 deg; joints [-12.917, -46.669, 112.704, 150.105, 51.247, -31.536, -355]
  MoveL 3764 to (-67.14, 2.34, -94.74) mm, rotated rx 42.04 ry 15.1 rz -114.75 deg; joints [-12.91, -46.588, 112.517, 150.07, 51.153, -31.471, -355]
  MoveL 3765 to (-66.92, 4.55, -94.92) mm, rotated rx 42.04 ry 15.1 rz -114.75 deg; joints [-12.904, -46.505, 112.323, 150.033, 51.056, -31.403, -355]
  MoveL 3766 to (-66.69, 6.77, -95.1) mm, rotated rx 42.04 ry 15.1 rz -114.75 deg; joints [-12.898, -46.421, 112.128, 149.995, 50.959, -31.335, -355]
  MoveL 3767 to (-66.49, 8.63, -95.34) mm, rotated rx 42.04 ry 15.1 rz -114.75 deg; joints [-12.896, -46.349, 111.963, 149.959, 50.878, -31.275, -355]
  MoveL 3768 to (-66.21, 11.29, -95.45) mm, rotated rx 42.04 ry 15.1 rz -114.75 deg; joints [-12.885, -46.248, 111.731, 149.919, 50.762, -31.196, -355]
  Set speed (1000.0 mm/s)
  MoveL 3769 to (-70.16, 56.42, -95.45) mm, rotated rx 42.04 ry 15.1 rz -114.75 deg; joints [-12.627, -45.013, 107.885, 149.106, 48.456, -29.584, -355]
  Set speed (1000.0 mm/s)
  MoveL 3770 to (-64.44, 56.92, -107.33) mm, rotated rx 42.04 ry 15.1 rz -114.75 deg; joints [-13.086, -44.596, 107.594, 148.598, 48.671, -29.432, -355]
  Set speed (100.0 mm/s)
  MoveL 3771 to (-61.94, 28.34, -107.33) mm, rotated rx 42.04 ry 15.1 rz -114.75 deg; joints [-13.255, -45.385, 110.042, 149.126, 50.129, -30.478, -355]
  MoveL 3772 to (-62.35, 26.67, -107.08) mm, rotated rx 42.04 ry 15.1 rz -114.75 deg; joints [-13.256, -45.465, 110.196, 149.157, 50.193, -30.527, -355]
  MoveL 3773 to (-62.8, 24.7, -107.02) mm, rotated rx 42.04 ry 15.1 rz -114.75 deg; joints [-13.266, -45.555, 110.375, 149.183, 50.271, -30.581, -355]
  MoveL 3774 to (-63.26, 22.7, -106.87) mm, rotated rx 42.04 ry 15.1 rz -114.75 deg; joints [-13.272, -45.648, 110.556, 149.213, 50.349, -30.637, -355]
  MoveL 3775 to (-63.83, 20.3, -106.74) mm, rotated rx 42.04 ry 15.1 rz -114.75 deg; joints [-13.282, -45.759, 110.773, 149.246, 50.442, -30.703, -355]
  MoveL 3776 to (-64.3, 18.22, -106.74) mm, rotated rx 42.04 ry 15.1 rz -114.75 deg; joints [-13.295, -45.854, 110.96, 149.269, 50.524, -30.758, -355]
  MoveL 3777 to (-64.81, 15.92, -106.58) mm, rotated rx 42.04 ry 15.1 rz -114.75 deg; joints [-13.303, -45.959, 111.167, 149.303, 50.614, -30.822, -355]
  MoveL 3778 to (-65.26, 13.98, -106.39) mm, rotated rx 42.04 ry 15.1 rz -114.75 deg; joints [-13.307, -46.048, 111.343, 149.333, 50.689, -30.877, -355]
  MoveL 3779 to (-65.72, 11.98, -106.3) mm, rotated rx 42.04 ry 15.1 rz -114.75 deg; joints [-13.316, -46.139, 111.523, 149.359, 50.767, -30.931, -355]
  MoveL 3780 to (-66.18, 9.9, -106.08) mm, rotated rx 42.04 ry 15.1 rz -114.75 deg; joints [-13.321, -46.234, 111.711, 149.393, 50.848, -30.99, -355]
  MoveL 3781 to (-66.64, 7.83, -105.93) mm, rotated rx 42.04 ry 15.1 rz -114.75 deg; joints [-13.327, -46.328, 111.896, 149.423, 50.928, -31.047, -355]
  MoveL 3782 to (-67.1, 5.77, -105.82) mm, rotated rx 42.04 ry 15.1 rz -114.75 deg; joints [-13.336, -46.421, 112.081, 149.45, 51.009, -31.103, -355]
  MoveL 3783 to (-67.55, 3.68, -105.65) mm, rotated rx 42.04 ry 15.1 rz -114.75 deg; joints [-13.342, -46.515, 112.268, 149.481, 51.091, -31.161, -355]
  MoveL 3784 to (-68, 1.6, -105.51) mm, rotated rx 42.04 ry 15.1 rz -114.75 deg; joints [-13.35, -46.608, 112.454, 149.51, 51.172, -31.218, -355]
  MoveL 3785 to (-68.47, -0.52, -105.44) mm, rotated rx 42.04 ry 15.1 rz -114.75 deg; joints [-13.361, -46.703, 112.642, 149.535, 51.255, -31.274, -355]
  MoveL 3786 to (-68.91, -2.61, -105.23) mm, rotated rx 42.04 ry 15.1 rz -114.75 deg; joints [-13.365, -46.796, 112.829, 149.567, 51.337, -31.333, -355]
  MoveL 3787 to (-69.35, -4.68, -105.11) mm, rotated rx 42.04 ry 15.1 rz -114.75 deg; joints [-13.374, -46.888, 113.013, 149.595, 51.418, -31.389, -355]
  MoveL 3788 to (-69.81, -6.8, -104.99) mm, rotated rx 42.04 ry 15.1 rz -114.75 deg; joints [-13.382, -46.982, 113.201, 149.622, 51.5, -31.446, -355]
  MoveL 3789 to (-70.05, -8.56, -104.78) mm, rotated rx 42.04 ry 15.1 rz -114.75 deg; joints [-13.385, -47.052, 113.356, 149.653, 51.574, -31.499, -355]
  MoveL 3790 to (-70.11, -10.03, -104.43) mm, rotated rx 42.04 ry 15.1 rz -114.75 deg; joints [-13.38, -47.103, 113.485, 149.691, 51.641, -31.552, -355]
  MoveL 3791 to (-69.98, -11.23, -103.9) mm, rotated rx 42.04 ry 15.1 rz -114.75 deg; joints [-13.366, -47.134, 113.591, 149.737, 51.702, -31.606, -355]
  MoveL 3792 to (-69.2, -9.9, -103.04) mm, rotated rx 42.04 ry 15.1 rz -114.75 deg; joints [-13.322, -47.05, 113.478, 149.777, 51.668, -31.607, -355]
  MoveL 3793 to (-69.54, -10.63, -103.04) mm, rotated rx 42.04 ry 15.1 rz -114.75 deg; joints [-13.327, -47.093, 113.544, 149.781, 51.69, -31.62, -355]
  MoveL 3794 to (-69.9, -11.23, -103.04) mm, rotated rx 42.04 ry 15.1 rz -114.75 deg; joints [-13.331, -47.134, 113.601, 149.783, 51.705, -31.628, -355]
  MoveL 3795 to (-70.3, -11.73, -103.04) mm, rotated rx 42.04 ry 15.1 rz -114.75 deg; joints [-13.334, -47.174, 113.649, 149.782, 51.712, -31.632, -355]
  MoveL 3796 to (-70.75, -12.22, -103.02) mm, rotated rx 42.04 ry 15.1 rz -114.75 deg; joints [-13.337, -47.217, 113.699, 149.782, 51.718, -31.635, -355]
  MoveL 3797 to (-71.28, -12.77, -102.98) mm, rotated rx 42.04 ry 15.1 rz -114.75 deg; joints [-13.339, -47.267, 113.754, 149.781, 51.723, -31.637, -355]
  MoveL 3798 to (-72.8, -14.21, -102.98) mm, rotated rx 42.04 ry 15.1 rz -114.75 deg; joints [-13.348, -47.405, 113.899, 149.773, 51.731, -31.638, -355]
  MoveL 3799 to (-73.12, -14.53, -102.96) mm, rotated rx 42.04 ry 15.1 rz -114.75 deg; joints [-13.35, -47.435, 113.931, 149.772, 51.734, -31.639, -355]
  MoveL 3800 to (-73.88, -15.25, -102.96) mm, rotated rx 42.04 ry 15.1 rz -114.75 deg; joints [-13.355, -47.504, 114.004, 149.768, 51.738, -31.639, -355]
  MoveL 3801 to (-74.24, -15.6, -102.96) mm, rotated rx 42.04 ry 15.1 rz -114.75 deg; joints [-13.357, -47.537, 114.039, 149.766, 51.74, -31.639, -355]
  MoveL 3802 to (-74.59, -15.94, -102.94) mm, rotated rx 42.04 ry 15.1 rz -114.75 deg; joints [-13.358, -47.569, 114.074, 149.765, 51.742, -31.64, -355]
  MoveL 3803 to (-74.92, -16.29, -102.91) mm, rotated rx 42.04 ry 15.1 rz -114.75 deg; joints [-13.359, -47.601, 114.109, 149.765, 51.745, -31.642, -355]
  MoveL 3804 to (-75.21, -16.61, -102.85) mm, rotated rx 42.04 ry 15.1 rz -114.75 deg; joints [-13.359, -47.629, 114.141, 149.767, 51.749, -31.645, -355]
  MoveL 3805 to (-75.53, -16.95, -102.81) mm, rotated rx 42.04 ry 15.1 rz -114.75 deg; joints [-13.36, -47.66, 114.176, 149.768, 51.752, -31.647, -355]
  MoveL 3806 to (-75.88, -17.3, -102.79) mm, rotated rx 42.04 ry 15.1 rz -114.75 deg; joints [-13.361, -47.693, 114.211, 149.767, 51.755, -31.647, -355]
  MoveL 3807 to (-76.25, -17.66, -102.78) mm, rotated rx 42.04 ry 15.1 rz -114.75 deg; joints [-13.363, -47.726, 114.246, 149.765, 51.757, -31.648, -355]
  MoveL 3808 to (-76.6, -18.01, -102.77) mm, rotated rx 42.04 ry 15.1 rz -114.75 deg; joints [-13.365, -47.759, 114.281, 149.764, 51.759, -31.649, -355]
  MoveL 3809 to (-76.92, -18.35, -102.73) mm, rotated rx 42.04 ry 15.1 rz -114.75 deg; joints [-13.366, -47.79, 114.316, 149.765, 51.763, -31.651, -355]
  MoveL 3810 to (-77.21, -18.68, -102.67) mm, rotated rx 42.04 ry 15.1 rz -114.75 deg; joints [-13.366, -47.818, 114.349, 149.767, 51.767, -31.654, -355]
  MoveL 3811 to (-77.51, -19.03, -102.62) mm, rotated rx 42.04 ry 15.1 rz -114.75 deg; joints [-13.366, -47.847, 114.383, 149.768, 51.771, -31.657, -355]
  MoveL 3812 to (-78.5, -20.06, -102.54) mm, rotated rx 42.04 ry 15.1 rz -114.75 deg; joints [-13.369, -47.942, 114.487, 149.768, 51.78, -31.661, -355]
  MoveL 3813 to (-79.42, -20.81, -102.66) mm, rotated rx 42.04 ry 15.1 rz -114.75 deg; joints [-13.38, -48.021, 114.562, 149.754, 51.778, -31.654, -355]
  MoveL 3814 to (-80.25, -21.25, -103) mm, rotated rx 42.04 ry 15.1 rz -114.75 deg; joints [-13.397, -48.084, 114.607, 149.727, 51.766, -31.635, -355]
  MoveL 3815 to (-80.64, -21.36, -103.25) mm, rotated rx 42.04 ry 15.1 rz -114.75 deg; joints [-13.408, -48.111, 114.619, 149.708, 51.756, -31.621, -355]
  MoveL 3816 to (-81, -21.4, -103.55) mm, rotated rx 42.04 ry 15.1 rz -114.75 deg; joints [-13.42, -48.133, 114.624, 149.686, 51.743, -31.604, -355]
  MoveL 3817 to (-81.67, -21.25, -104.31) mm, rotated rx 42.04 ry 15.1 rz -114.75 deg; joints [-13.451, -48.166, 114.612, 149.632, 51.71, -31.562, -355]
  MoveL 3818 to (-82.26, -20.8, -105.27) mm, rotated rx 42.04 ry 15.1 rz -114.75 deg; joints [-13.488, -48.183, 114.571, 149.564, 51.667, -31.508, -355]
  MoveL 3819 to (-83.19, -19.01, -107.84) mm, rotated rx 42.04 ry 15.1 rz -114.75 deg; joints [-13.582, -48.172, 114.401, 149.389, 51.55, -31.364, -355]
  MoveL 3820 to (-83.54, -16.69, -110.45) mm, rotated rx 42.04 ry 15.1 rz -114.75 deg; joints [-13.674, -48.107, 114.177, 149.214, 51.432, -31.219, -355]
  MoveL 3821 to (-83.4, -15.58, -111.48) mm, rotated rx 42.04 ry 15.1 rz -114.75 deg; joints [-13.708, -48.059, 114.067, 149.148, 51.387, -31.163, -355]
  MoveL 3822 to (-83.06, -14.5, -112.32) mm, rotated rx 42.04 ry 15.1 rz -114.75 deg; joints [-13.735, -47.999, 113.959, 149.096, 51.351, -31.12, -355]
  MoveL 3823 to (-82.5, -13.45, -112.97) mm, rotated rx 42.04 ry 15.1 rz -114.75 deg; joints [-13.755, -47.929, 113.854, 149.058, 51.325, -31.088, -355]
  MoveL 3824 to (-81.75, -12.43, -113.44) mm, rotated rx 42.04 ry 15.1 rz -114.75 deg; joints [-13.767, -47.847, 113.75, 149.035, 51.308, -31.067, -355]
  MoveL 3825 to (-80.78, -11.44, -113.72) mm, rotated rx 42.04 ry 15.1 rz -114.75 deg; joints [-13.771, -47.755, 113.648, 149.025, 51.3, -31.059, -355]
  MoveL 3826 to (-79.61, -10.48, -113.81) mm, rotated rx 42.04 ry 15.1 rz -114.75 deg; joints [-13.768, -47.652, 113.548, 149.03, 51.302, -31.062, -355]
  MoveL 3827 to (-77.07, -8.6, -113.81) mm, rotated rx 42.04 ry 15.1 rz -114.75 deg; joints [-13.755, -47.437, 113.35, 149.053, 51.314, -31.079, -355]
  MoveL 3828 to (-76.63, -8.26, -113.83) mm, rotated rx 42.04 ry 15.1 rz -114.75 deg; joints [-13.753, -47.4, 113.314, 149.056, 51.315, -31.081, -355]
  MoveL 3829 to (-76.14, -7.87, -113.86) mm, rotated rx 42.04 ry 15.1 rz -114.75 deg; joints [-13.752, -47.358, 113.273, 149.058, 51.316, -31.083, -355]
  MoveL 3830 to (-75.57, -7.38, -113.96) mm, rotated rx 42.04 ry 15.1 rz -114.75 deg; joints [-13.752, -47.306, 113.221, 149.057, 51.315, -31.082, -355]
  MoveL 3831 to (-75.09, -6.99, -113.99) mm, rotated rx 42.04 ry 15.1 rz -114.75 deg; joints [-13.751, -47.264, 113.18, 149.059, 51.316, -31.083, -355]
  MoveL 3832 to (-74.65, -6.66, -114.01) mm, rotated rx 42.04 ry 15.1 rz -114.75 deg; joints [-13.749, -47.227, 113.145, 149.062, 51.317, -31.085, -355]
  MoveL 3833 to (-74.25, -6.35, -114.02) mm, rotated rx 42.04 ry 15.1 rz -114.75 deg; joints [-13.747, -47.193, 113.112, 149.065, 51.318, -31.087, -355]
  MoveL 3834 to (-73.89, -6.07, -114.03) mm, rotated rx 42.04 ry 15.1 rz -114.75 deg; joints [-13.746, -47.162, 113.082, 149.067, 51.319, -31.089, -355]
  MoveL 3835 to (-72.24, -4.84, -114.04) mm, rotated rx 42.04 ry 15.1 rz -114.75 deg; joints [-13.738, -47.022, 112.952, 149.081, 51.325, -31.099, -355]
  MoveL 3836 to (-71.84, -4.52, -114.08) mm, rotated rx 42.04 ry 15.1 rz -114.75 deg; joints [-13.737, -46.987, 112.918, 149.082, 51.326, -31.099, -355]
  MoveL 3837 to (-71.48, -4.21, -114.13) mm, rotated rx 42.04 ry 15.1 rz -114.75 deg; joints [-13.737, -46.955, 112.885, 149.082, 51.325, -31.099, -355]
  MoveL 3838 to (-71.15, -3.89, -114.2) mm, rotated rx 42.04 ry 15.1 rz -114.75 deg; joints [-13.738, -46.925, 112.852, 149.08, 51.323, -31.097, -355]
  MoveL 3839 to (-70.81, -3.54, -114.26) mm, rotated rx 42.04 ry 15.1 rz -114.75 deg; joints [-13.738, -46.892, 112.816, 149.079, 51.32, -31.095, -355]
  MoveL 3840 to (-70.44, -3.13, -114.29) mm, rotated rx 42.04 ry 15.1 rz -114.75 deg; joints [-13.736, -46.857, 112.775, 149.078, 51.315, -31.092, -355]
  MoveL 3841 to (-70.06, -2.58, -114.3) mm, rotated rx 42.04 ry 15.1 rz -114.75 deg; joints [-13.733, -46.816, 112.722, 149.077, 51.304, -31.085, -355]
  MoveL 3842 to (-69.68, -1.9, -114.3) mm, rotated rx 42.04 ry 15.1 rz -114.75 deg; joints [-13.728, -46.772, 112.659, 149.075, 51.286, -31.074, -355]
  MoveL 3843 to (-71.32, -2.95, -115.86) mm, rotated rx 42.04 ry 15.1 rz -114.75 deg; joints [-13.798, -46.896, 112.752, 148.978, 51.275, -31.023, -355]
  MoveL 3844 to (-70.55, -0.71, -115.99) mm, rotated rx 42.04 ry 15.1 rz -114.75 deg; joints [-13.789, -46.779, 112.549, 148.954, 51.199, -30.97, -355]
  MoveL 3845 to (-69.81, 1.4, -116.1) mm, rotated rx 42.04 ry 15.1 rz -114.75 deg; joints [-13.779, -46.667, 112.356, 148.932, 51.128, -30.921, -355]
  MoveL 3846 to (-69.12, 3.44, -116.26) mm, rotated rx 42.04 ry 15.1 rz -114.75 deg; joints [-13.772, -46.56, 112.17, 148.907, 51.058, -30.871, -355]
  MoveL 3847 to (-68.42, 5.46, -116.37) mm, rotated rx 42.04 ry 15.1 rz -114.75 deg; joints [-13.763, -46.453, 111.985, 148.886, 50.99, -30.824, -355]
  MoveL 3848 to (-67.72, 7.47, -116.48) mm, rotated rx 42.04 ry 15.1 rz -114.75 deg; joints [-13.754, -46.347, 111.801, 148.864, 50.921, -30.776, -355]
  MoveL 3849 to (-67.03, 9.5, -116.7) mm, rotated rx 42.04 ry 15.1 rz -114.75 deg; joints [-13.749, -46.24, 111.614, 148.836, 50.852, -30.725, -355]
  MoveL 3850 to (-66.33, 11.51, -116.92) mm, rotated rx 42.04 ry 15.1 rz -114.75 deg; joints [-13.745, -46.133, 111.427, 148.808, 50.783, -30.674, -355]
  MoveL 3851 to (-65.62, 13.53, -117.04) mm, rotated rx 42.04 ry 15.1 rz -114.75 deg; joints [-13.736, -46.025, 111.242, 148.785, 50.714, -30.626, -355]
  MoveL 3852 to (-64.9, 15.54, -117.04) mm, rotated rx 42.04 ry 15.1 rz -114.75 deg; joints [-13.723, -45.918, 111.059, 148.769, 50.646, -30.581, -355]
  MoveL 3853 to (-64.19, 17.55, -117.15) mm, rotated rx 42.04 ry 15.1 rz -114.75 deg; joints [-13.714, -45.81, 110.873, 148.746, 50.577, -30.533, -355]
  MoveL 3854 to (-63.46, 19.59, -117.35) mm, rotated rx 42.04 ry 15.1 rz -114.75 deg; joints [-13.709, -45.701, 110.683, 148.718, 50.508, -30.481, -355]
  MoveL 3855 to (-62.79, 21.48, -117.53) mm, rotated rx 42.04 ry 15.1 rz -114.75 deg; joints [-13.703, -45.598, 110.507, 148.693, 50.443, -30.434, -355]
  MoveL 3856 to (-62.16, 23.23, -117.75) mm, rotated rx 42.04 ry 15.1 rz -114.75 deg; joints [-13.701, -45.504, 110.343, 148.666, 50.384, -30.389, -355]
  MoveL 3857 to (-61.5, 25.08, -117.84) mm, rotated rx 42.04 ry 15.1 rz -114.75 deg; joints [-13.692, -45.404, 110.171, 148.646, 50.32, -30.344, -355]
  MoveL 3858 to (-60.79, 27.05, -117.85) mm, rotated rx 42.04 ry 15.1 rz -114.75 deg; joints [-13.68, -45.299, 109.99, 148.628, 50.252, -30.298, -355]
  MoveL 3859 to (-59.86, 29.6, -117.95) mm, rotated rx 42.04 ry 15.1 rz -114.75 deg; joints [-13.667, -45.161, 109.753, 148.6, 50.165, -30.237, -355]
  MoveL 3860 to (-59.16, 31.51, -118.16) mm, rotated rx 42.04 ry 15.1 rz -114.75 deg; joints [-13.663, -45.056, 109.573, 148.572, 50.1, -30.188, -355]
  MoveL 3861 to (-58.39, 33.57, -118.36) mm, rotated rx 42.04 ry 15.1 rz -114.75 deg; joints [-13.658, -44.942, 109.379, 148.544, 50.03, -30.136, -355]
  MoveL 3862 to (-57.67, 35.46, -118.65) mm, rotated rx 42.04 ry 15.1 rz -114.75 deg; joints [-13.657, -44.837, 109.199, 148.512, 49.967, -30.086, -355]
  MoveL 3863 to (-56.99, 37.32, -118.78) mm, rotated rx 42.04 ry 15.1 rz -114.75 deg; joints [-13.65, -44.735, 109.024, 148.488, 49.903, -30.039, -355]
  MoveL 3864 to (-56.28, 39.29, -118.79) mm, rotated rx 42.04 ry 15.1 rz -114.75 deg; joints [-13.638, -44.629, 108.84, 148.469, 49.834, -29.992, -355]
  MoveL 3865 to (-55.63, 40.94, -119.02) mm, rotated rx 42.04 ry 15.1 rz -114.75 deg; joints [-13.636, -44.535, 108.682, 148.442, 49.779, -29.949, -355]
  Set speed (1000.0 mm/s)
  MoveL 3866 to (-57.9, 66.9, -119.02) mm, rotated rx 42.04 ry 15.1 rz -114.75 deg; joints [-13.477, -43.809, 106.442, 147.946, 48.454, -28.973, -355]
  Set speed (1000.0 mm/s)
  MoveL 3867 to (-51.39, 67.47, -130.21) mm, rotated rx 42.04 ry 15.1 rz -114.75 deg; joints [-13.901, -43.342, 106.117, 147.491, 48.679, -28.855, -355]
  Set speed (100.0 mm/s)
  MoveL 3868 to (-49.64, 47.38, -130.21) mm, rotated rx 42.04 ry 15.1 rz -114.75 deg; joints [-14.03, -43.903, 107.855, 147.878, 49.704, -29.622, -355]
  MoveL 3869 to (-50.6, 45.47, -130.21) mm, rotated rx 42.04 ry 15.1 rz -114.75 deg; joints [-14.042, -44.022, 108.038, 147.891, 49.761, -29.661, -355]
  MoveL 3870 to (-51.63, 43.49, -130.11) mm, rotated rx 42.04 ry 15.1 rz -114.75 deg; joints [-14.052, -44.148, 108.23, 147.909, 49.819, -29.702, -355]
  MoveL 3871 to (-52.75, 41.43, -129.82) mm, rotated rx 42.04 ry 15.1 rz -114.75 deg; joints [-14.054, -44.283, 108.434, 147.937, 49.878, -29.748, -355]
  MoveL 3872 to (-53.82, 39.45, -129.47) mm, rotated rx 42.04 ry 15.1 rz -114.75 deg; joints [-14.054, -44.414, 108.63, 147.966, 49.933, -29.794, -355]
  MoveL 3873 to (-54.78, 37.62, -129.28) mm, rotated rx 42.04 ry 15.1 rz -114.75 deg; joints [-14.059, -44.531, 108.808, 147.987, 49.986, -29.834, -355]
  MoveL 3874 to (-55.67, 35.88, -129.15) mm, rotated rx 42.04 ry 15.1 rz -114.75 deg; joints [-14.066, -44.642, 108.976, 148.005, 50.036, -29.871, -355]
  MoveL 3875 to (-56.61, 34.06, -129.1) mm, rotated rx 42.04 ry 15.1 rz -114.75 deg; joints [-14.076, -44.757, 109.151, 148.019, 50.09, -29.907, -355]
  MoveL 3876 to (-57.57, 32.15, -129.07) mm, rotated rx 42.04 ry 15.1 rz -114.75 deg; joints [-14.088, -44.876, 109.333, 148.032, 50.146, -29.944, -355]
  MoveL 3877 to (-58.53, 30.26, -128.96) mm, rotated rx 42.04 ry 15.1 rz -114.75 deg; joints [-14.096, -44.995, 109.515, 148.05, 50.2, -29.983, -355]
  MoveL 3878 to (-59.58, 28.22, -128.7) mm, rotated rx 42.04 ry 15.1 rz -114.75 deg; joints [-14.1, -45.124, 109.712, 148.075, 50.259, -30.028, -355]
  MoveL 3879 to (-60.66, 26.08, -128.51) mm, rotated rx 42.04 ry 15.1 rz -114.75 deg; joints [-14.108, -45.259, 109.918, 148.097, 50.321, -30.074, -355]
  MoveL 3880 to (-61.71, 24, -128.31) mm, rotated rx 42.04 ry 15.1 rz -114.75 deg; joints [-14.114, -45.39, 110.118, 148.12, 50.381, -30.118, -355]
  MoveL 3881 to (-62.67, 22.09, -128.2) mm, rotated rx 42.04 ry 15.1 rz -114.75 deg; joints [-14.123, -45.509, 110.299, 148.137, 50.436, -30.157, -355]
  MoveL 3882 to (-64.55, 18.31, -127.92) mm, rotated rx 42.04 ry 15.1 rz -114.75 deg; joints [-14.138, -45.745, 110.659, 148.172, 50.544, -30.234, -355]
  MoveL 3883 to (-65.53, 16.37, -127.86) mm, rotated rx 42.04 ry 15.1 rz -114.75 deg; joints [-14.149, -45.867, 110.843, 148.186, 50.6, -30.272, -355]
  MoveL 3884 to (-66.47, 14.45, -127.64) mm, rotated rx 42.04 ry 15.1 rz -114.75 deg; joints [-14.153, -45.986, 111.025, 148.209, 50.655, -30.313, -355]
  MoveL 3885 to (-67.4, 12.56, -127.48) mm, rotated rx 42.04 ry 15.1 rz -114.75 deg; joints [-14.16, -46.103, 111.205, 148.227, 50.709, -30.352, -355]
  MoveL 3886 to (-68.32, 10.66, -127.29) mm, rotated rx 42.04 ry 15.1 rz -114.75 deg; joints [-14.166, -46.22, 111.385, 148.247, 50.764, -30.392, -355]
  MoveL 3887 to (-69.29, 8.71, -127.2) mm, rotated rx 42.04 ry 15.1 rz -114.75 deg; joints [-14.176, -46.341, 111.568, 148.262, 50.819, -30.43, -355]
  MoveL 3888 to (-70.28, 6.66, -127.07) mm, rotated rx 42.04 ry 15.1 rz -114.75 deg; joints [-14.185, -46.467, 111.76, 148.279, 50.878, -30.471, -355]
  MoveL 3889 to (-71.14, 4.97, -127.01) mm, rotated rx 42.04 ry 15.1 rz -114.75 deg; joints [-14.195, -46.573, 111.919, 148.29, 50.924, -30.502, -355]
  MoveL 3890 to (-70.55, 4.67, -126.13) mm, rotated rx 42.04 ry 15.1 rz -114.75 deg; joints [-14.161, -46.552, 111.948, 148.352, 50.96, -30.551, -355]
  MoveL 3891 to (-70.23, 4.83, -125.71) mm, rotated rx 42.04 ry 15.1 rz -114.75 deg; joints [-14.143, -46.529, 111.935, 148.377, 50.964, -30.566, -355]
  MoveL 3892 to (-70.16, 4.82, -125.44) mm, rotated rx 42.04 ry 15.1 rz -114.75 deg; joints [-14.132, -46.527, 111.939, 148.393, 50.967, -30.575, -355]
  MoveL 3893 to (-70.42, 4.62, -125.32) mm, rotated rx 42.04 ry 15.1 rz -114.75 deg; joints [-14.129, -46.55, 111.962, 148.397, 50.966, -30.577, -355]
  MoveL 3894 to (-70.79, 4.36, -125.26) mm, rotated rx 42.04 ry 15.1 rz -114.75 deg; joints [-14.128, -46.581, 111.99, 148.397, 50.964, -30.575, -355]
  MoveL 3895 to (-71.27, 4.07, -125.23) mm, rotated rx 42.04 ry 15.1 rz -114.75 deg; joints [-14.129, -46.62, 112.024, 148.393, 50.959, -30.571, -355]
  MoveL 3896 to (-71.86, 3.7, -125.19) mm, rotated rx 42.04 ry 15.1 rz -114.75 deg; joints [-14.13, -46.668, 112.065, 148.389, 50.954, -30.566, -355]
  MoveL 3897 to (-72.41, 3.38, -125.16) mm, rotated rx 42.04 ry 15.1 rz -114.75 deg; joints [-14.132, -46.711, 112.101, 148.384, 50.948, -30.56, -355]
  MoveL 3898 to (-72.86, 3.13, -125.16) mm, rotated rx 42.04 ry 15.1 rz -114.75 deg; joints [-14.133, -46.747, 112.13, 148.379, 50.943, -30.555, -355]
  MoveL 3899 to (-73.28, 2.88, -125.15) mm, rotated rx 42.04 ry 15.1 rz -114.75 deg; joints [-14.135, -46.781, 112.158, 148.375, 50.938, -30.551, -355]
  MoveL 3900 to (-74.16, 2.32, -125.07) mm, rotated rx 42.04 ry 15.1 rz -114.75 deg; joints [-14.136, -46.852, 112.221, 148.37, 50.93, -30.544, -355]
  MoveL 3901 to (-74.63, 2.02, -125.02) mm, rotated rx 42.04 ry 15.1 rz -114.75 deg; joints [-14.136, -46.891, 112.254, 148.368, 50.927, -30.541, -355]
  MoveL 3902 to (-75.05, 1.73, -124.95) mm, rotated rx 42.04 ry 15.1 rz -114.75 deg; joints [-14.135, -46.926, 112.287, 148.367, 50.924, -30.539, -355]
  MoveL 3903 to (-75.43, 1.46, -124.88) mm, rotated rx 42.04 ry 15.1 rz -114.75 deg; joints [-14.134, -46.958, 112.317, 148.368, 50.922, -30.538, -355]
  MoveL 3904 to (-75.82, 1.2, -124.82) mm, rotated rx 42.04 ry 15.1 rz -114.75 deg; joints [-14.134, -46.99, 112.346, 148.367, 50.919, -30.536, -355]
  MoveL 3905 to (-76.23, 0.94, -124.79) mm, rotated rx 42.04 ry 15.1 rz -114.75 deg; joints [-14.135, -47.023, 112.374, 148.364, 50.915, -30.533, -355]
  MoveL 3906 to (-76.68, 0.68, -124.77) mm, rotated rx 42.04 ry 15.1 rz -114.75 deg; joints [-14.136, -47.059, 112.404, 148.36, 50.911, -30.528, -355]
  MoveL 3907 to (-79.87, -1.12, -124.77) mm, rotated rx 42.04 ry 15.1 rz -114.75 deg; joints [-14.149, -47.311, 112.606, 148.323, 50.871, -30.488, -355]
  MoveL 3908 to (-81.34, -1.82, -124.79) mm, rotated rx 42.04 ry 15.1 rz -114.75 deg; joints [-14.156, -47.423, 112.688, 148.302, 50.847, -30.465, -355]
  MoveL 3909 to (-81.89, -1.98, -124.81) mm, rotated rx 42.04 ry 15.1 rz -114.75 deg; joints [-14.158, -47.462, 112.71, 148.292, 50.833, -30.452, -355]
  MoveL 3910 to (-82.33, -2.03, -124.85) mm, rotated rx 42.04 ry 15.1 rz -114.75 deg; joints [-14.16, -47.49, 112.72, 148.282, 50.818, -30.439, -355]
  MoveL 3911 to (-82.67, -1.97, -124.89) mm, rotated rx 42.04 ry 15.1 rz -114.75 deg; joints [-14.161, -47.509, 112.72, 148.272, 50.802, -30.426, -355]
  MoveL 3912 to (-82.8, -1.91, -124.92) mm, rotated rx 42.04 ry 15.1 rz -114.75 deg; joints [-14.162, -47.515, 112.716, 148.268, 50.794, -30.419, -355]
  MoveL 3913 to (-82.91, -1.82, -124.94) mm, rotated rx 42.04 ry 15.1 rz -114.75 deg; joints [-14.162, -47.518, 112.71, 148.263, 50.786, -30.412, -355]
  MoveL 3914 to (-83, -1.72, -124.97) mm, rotated rx 42.04 ry 15.1 rz -114.75 deg; joints [-14.163, -47.52, 112.702, 148.258, 50.778, -30.405, -355]
  MoveL 3915 to (-83.07, -1.59, -125) mm, rotated rx 42.04 ry 15.1 rz -114.75 deg; joints [-14.163, -47.52, 112.692, 148.253, 50.769, -30.398, -355]
  MoveL 3916 to (-83.14, -1.29, -125.06) mm, rotated rx 42.04 ry 15.1 rz -114.75 deg; joints [-14.164, -47.515, 112.666, 148.244, 50.752, -30.384, -355]
  MoveL 3917 to (-83.1, -0.49, -125.19) mm, rotated rx 42.04 ry 15.1 rz -114.75 deg; joints [-14.163, -47.486, 112.597, 148.227, 50.717, -30.357, -355]
  MoveL 3918 to (-82.84, 0.48, -125.33) mm, rotated rx 42.04 ry 15.1 rz -114.75 deg; joints [-14.162, -47.438, 112.508, 148.211, 50.682, -30.329, -355]
  MoveL 3919 to (-81.94, 2.64, -125.6) mm, rotated rx 42.04 ry 15.1 rz -114.75 deg; joints [-14.158, -47.313, 112.307, 148.183, 50.617, -30.279, -355]
  MoveL 3920 to (-80.88, 4.81, -125.84) mm, rotated rx 42.04 ry 15.1 rz -114.75 deg; joints [-14.152, -47.178, 112.103, 148.16, 50.558, -30.235, -355]
  MoveL 3921 to (-56.65, 53.05, -130.92) mm, rotated rx 42.04 ry 15.1 rz -114.75 deg; joints [-14.023, -44.128, 107.47, 147.607, 49.186, -29.197, -355]
  MoveL 3922 to (-54.93, 56.48, -131.28) mm, rotated rx 42.04 ry 15.1 rz -114.75 deg; joints [-14.014, -43.91, 107.134, 147.563, 49.084, -29.117, -355]
  MoveL 3923 to (-53.09, 59.74, -131.7) mm, rotated rx 42.04 ry 15.1 rz -114.75 deg; joints [-14.008, -43.691, 106.808, 147.52, 48.993, -29.045, -355]
  MoveL 3924 to (-52.13, 60.88, -131.91) mm, rotated rx 42.04 ry 15.1 rz -114.75 deg; joints [-14.009, -43.595, 106.688, 147.508, 48.972, -29.027, -355]
  MoveL 3925 to (-51.68, 61.19, -132) mm, rotated rx 42.04 ry 15.1 rz -114.75 deg; joints [-14.01, -43.558, 106.651, 147.507, 48.974, -29.027, -355]
  MoveL 3926 to (-51.46, 61.26, -132.05) mm, rotated rx 42.04 ry 15.1 rz -114.75 deg; joints [-14.012, -43.542, 106.641, 147.508, 48.978, -29.03, -355]
  MoveL 3927 to (-51.25, 61.26, -132.09) mm, rotated rx 42.04 ry 15.1 rz -114.75 deg; joints [-14.013, -43.53, 106.636, 147.509, 48.985, -29.035, -355]
  MoveL 3928 to (-51.05, 61.2, -132.13) mm, rotated rx 42.04 ry 15.1 rz -114.75 deg; joints [-14.015, -43.52, 106.638, 147.513, 48.995, -29.042, -355]
  MoveL 3929 to (-50.86, 61.06, -132.16) mm, rotated rx 42.04 ry 15.1 rz -114.75 deg; joints [-14.017, -43.513, 106.646, 147.517, 49.008, -29.051, -355]
  MoveL 3930 to (-50.69, 60.85, -132.19) mm, rotated rx 42.04 ry 15.1 rz -114.75 deg; joints [-14.019, -43.51, 106.661, 147.523, 49.025, -29.063, -355]
  MoveL 3931 to (-50.52, 60.55, -132.22) mm, rotated rx 42.04 ry 15.1 rz -114.75 deg; joints [-14.022, -43.51, 106.684, 147.53, 49.045, -29.078, -355]
  MoveL 3932 to (-50.02, 58.41, -132.26) mm, rotated rx 42.04 ry 15.1 rz -114.75 deg; joints [-14.038, -43.551, 106.863, 147.575, 49.164, -29.168, -355]
  MoveL 3933 to (-49.77, 56.34, -132.26) mm, rotated rx 42.04 ry 15.1 rz -114.75 deg; joints [-14.051, -43.605, 107.041, 147.616, 49.273, -29.25, -355]
  MoveL 3934 to (-49.77, 52.53, -132.31) mm, rotated rx 42.04 ry 15.1 rz -114.75 deg; joints [-14.078, -43.729, 107.375, 147.68, 49.456, -29.384, -355]
  MoveL 3935 to (-50.54, 49.07, -132.42) mm, rotated rx 42.04 ry 15.1 rz -114.75 deg; joints [-14.105, -43.888, 107.69, 147.718, 49.594, -29.481, -355]
  MoveL 3936 to (-53.25, 43.66, -132.72) mm, rotated rx 42.04 ry 15.1 rz -114.75 deg; joints [-14.153, -44.223, 108.205, 147.741, 49.758, -29.583, -355]
  MoveL 3937 to (-54.73, 41.82, -132.85) mm, rotated rx 42.04 ry 15.1 rz -114.75 deg; joints [-14.171, -44.37, 108.389, 147.737, 49.793, -29.6, -355]
  MoveL 3938 to (-77.59, 15.62, -134.71) mm, rotated rx 42.04 ry 15.1 rz -114.75 deg; joints [-14.432, -46.577, 110.999, 147.602, 50.194, -29.756, -355]
  MoveL 3939 to (-79.53, 13.37, -134.87) mm, rotated rx 42.04 ry 15.1 rz -114.75 deg; joints [-14.454, -46.766, 111.219, 147.588, 50.226, -29.767, -355]
  MoveL 3940 to (-81.61, 10.27, -135.12) mm, rotated rx 42.04 ry 15.1 rz -114.75 deg; joints [-14.487, -46.99, 111.512, 147.58, 50.292, -29.8, -355]
  MoveL 3941 to (-82.14, 8.89, -135.26) mm, rotated rx 42.04 ry 15.1 rz -114.75 deg; joints [-14.502, -47.066, 111.636, 147.583, 50.336, -29.826, -355]
  MoveL 3942 to (-82.18, 8.34, -135.33) mm, rotated rx 42.04 ry 15.1 rz -114.75 deg; joints [-14.509, -47.085, 111.682, 147.587, 50.36, -29.842, -355]
  MoveL 3943 to (-82.13, 8.12, -135.36) mm, rotated rx 42.04 ry 15.1 rz -114.75 deg; joints [-14.512, -47.089, 111.699, 147.589, 50.372, -29.85, -355]
  MoveL 3944 to (-82.03, 7.94, -135.4) mm, rotated rx 42.04 ry 15.1 rz -114.75 deg; joints [-14.514, -47.088, 111.713, 147.592, 50.385, -29.858, -355]
  MoveL 3945 to (-81.87, 7.8, -135.43) mm, rotated rx 42.04 ry 15.1 rz -114.75 deg; joints [-14.517, -47.083, 111.722, 147.596, 50.397, -29.867, -355]
  MoveL 3946 to (-81.66, 7.7, -135.47) mm, rotated rx 42.04 ry 15.1 rz -114.75 deg; joints [-14.519, -47.073, 111.726, 147.6, 50.41, -29.876, -355]
  MoveL 3947 to (-81.38, 7.66, -135.5) mm, rotated rx 42.04 ry 15.1 rz -114.75 deg; joints [-14.52, -47.057, 111.725, 147.605, 50.422, -29.886, -355]
